// TIA Portal project "Trabajo_plantilla" (V14)
// Plantilla para la realización de la parte de programación de la asignatura de Automatización

(* hardware
DEVICE "S71500/ET200MP station_1"  S7-1500 station
   slot 0: "Perfil soporte_0"  Rack  6ES7 590-1***0-0AA0
   slot 1: "FINAL"  CPU 1516F-3 PN/DP  6ES7 516-3FN00-0AB0  V1.8
      slot 3: "Display de la CPU_1"  6ES7591-1BA00-0AA0
   slot 2: "DI 32x24VDC HF_1"  DI 32x24VDC HF  6ES7 521-1BL00-0AB0  V2.1
   slot 3: "DQ 16x24VDC/0.5A HF_1"  DQ 16x24VDC/0.5A HF  6ES7 522-1BH01-0AB0  V1.0
   slot 4: "AI 8xU/I/RTD/TC ST_1"  AI 8xU/I/RTD/TC ST  6ES7 531-7KF00-0AB0  V2.1
   slot 5: "AQ 4xU/I ST_1"  AQ 4xU/I ST  6ES7 532-5HD00-0AB0  V2.1
   slot 6: "DI 32x24VDC HF_2"  DI 32x24VDC HF  6ES7 521-1BL00-0AB0  V2.1
*)

// ===== PLC "FINAL"  CPU 1516F-3 PN/DP =====

VAR_GLOBAL   // PLC tag table "Variables maq_tem_HORNO"
   "Rearme_HORNO" AT %E2.1 : Bool;
   "Emer_HORNO" AT %E2.2 : Bool;
   "T_Cinta_Horno" AT %T8 : Timer;
   "Temperatura_REAL_HORNO" AT %MD11 : Real;
   "Temperatura_SENSOR_HORNO" AT %EW10 : Int;
   "Aviso_Foco_OK_HORNO" AT %M2.2 : Bool;
   "Aviso_error_sincrono_EXT_HORNO" AT %M2.4 : Bool;
   "Aviso_error_sensor_EXT_HORNO" AT %M2.5 : Bool;
   "S_piezas_cargadas_HORNO" AT %E2.3 : Bool;
   "S_piezas_descargadas_HORNO" AT %E2.4 : Bool;
   "MOV_CINTA_HORNO" AT %A0.0 : Bool;
   "FOCO_HORNO" AT %A2.2 : Bool;
   "MODO_FOCO" AT %E2.5 : Bool;
   "Aviso_Standby_HORNO" AT %M2.6 : Bool;
   "START_HORNO" AT %E2.0 : Bool;
END_VAR

VAR_GLOBAL   // PLC tag table "Variables CONFORMADORA"
   "Emer_CONFOR" AT %E1.2 : Bool;
   "Rearme_CONFOR" AT %E1.1 : Bool;
   "S_final_CONFOR" AT %E1.3 : Bool;
   "T_compresion_CONFOR" AT %T1 : Timer;
   "T_descompresion_CONFOR" AT %T2 : Timer;
   "Fuerza_SENSOR_CONFOR" AT %EW12 : Int;
   "Aviso_Pieza_Cargada_CONFOR" AT %E1.4 : Bool;
   "Aviso_Pieza_Desargada_CONFOR" AT %E1.5 : Bool;
   "Aviso_Standby_CONFOR" AT %M1.0 : Bool;
   "Aviso_error_sincrono_EXT_CONFOR" AT %M1.1 : Bool;
   "Aviso_error_sensor_EXT_CONFOR" AT %M1.2 : Bool;
   "Fuerza_REAL_CONFOR" AT %MD7 : Real;
   "COMPRIMIR_CONFOR" AT %A1.0 : Bool;
   "DESCOMPRIMIR_CONFOR" AT %A1.1 : Bool;
   "START_CONFOR" AT %E1.0 : Bool;
END_VAR

VAR_GLOBAL   // PLC tag table "Variables ROBOT"
   "START_ROBOT" AT %E5.0 : Bool;
   "EMER_ROBOT" AT %E5.1 : Bool;
   "Rearme_ROBOT" AT %E5.3 : Bool;
   "Tlimite_ROBOT" AT %T11 : Timer;
   "T_espera_ROBOT" AT %T12 : Timer;
   "MODO_M1_Descarga_ROBOT" AT %M5.0 : Bool;
   "MODO_M2_Carga_ROBOT" AT %M5.1 : Bool;
   "Zona_descarga_libre" AT %M5.2 : Bool;
   "Aviso_error_sincrono_ROBOT" AT %M5.3 : Bool;
   "Aviso_error_asincrono_ROBOT" AT %M5.4 : Bool;
   "Aviso_emergencia_ROBOT" AT %M5.5 : Bool;
   "Aviso_de_standby_ROBOT" AT %M5.6 : Bool;
   "SB_pieza_esperando" AT %E5.4 : Bool;   // Variables brazo robot
   "SB_pinza_llena_brazo" AT %E5.5 : Bool;
   "SB_llegada_Carga" AT %E5.6 : Bool;
   "SB_llegada_Descarga" AT %E5.7 : Bool;
   "SB_llegada_a_reposo" AT %E5.2 : Bool;
   "Mov1" AT %A5.0 : Bool;
   "Mov2" AT %A5.1 : Bool;
   "Mov3" AT %A5.2 : Bool;
   "Act1" AT %A5.3 : Bool;
   "Act2" AT %A5.4 : Bool;
   "X_Espera_maquina_libre" AT %M5.7 : Bool;
   "Aviso_STDBY_ROBOT" AT %M6.0 : Bool;
   "Aviso_maquina_libre" AT %M6.1 : Bool;
END_VAR

VAR_GLOBAL   // PLC tag table "Variables maq_tem_TUNEL"
   "Rearme_TUNEL" AT %E3.1 : Bool;
   "Emer_TUNEL" AT %E3.2 : Bool;
   "T_Cinta_Tunel" AT %T9 : Timer;
   "Temperatura_REAL_TUNEL" AT %MD15 : Real;
   "Temperatura_SENSOR_TUNEL" AT %EW8 : Int;
   "Aviso_Foco_OK_TUNEL" AT %M3.1 : Bool;
   "Aviso_error_sincrono_EXT_TUNEL" AT %M3.3 : Bool;
   "Aviso_error_sensor_EXT_TUNEL" AT %M3.4 : Bool;
   "S_piezas_descargadas_TUNEL" AT %E3.4 : Bool;
   "MOV_CINTA_TUNEL" AT %A3.0 : Bool;
   "FOCO_TUNEL" AT %A3.1 : Bool;
   "MODO_FOCO_TUNEL" AT %E3.5 : Bool;
   "Aviso_Standby_TUNEL" AT %M3.5 : Bool;
   "START_TUNEL" AT %E3.0 : Bool;
   "S_piezas_cargadas_TUNEL" AT %E3.3 : Bool;
END_VAR

VAR_GLOBAL   // PLC tag table "Variables PULIDORA"
   "Spieza_PULI" AT %E6.0 : Bool;
   "S_F_Mov_Cab" AT %E6.1 : Bool;
   "S_F_Mov_Cab2" AT %E6.2 : Bool;
   "S_F_Acercar" AT %E6.3 : Bool;
   "S_F_Pulido1" AT %E6.4 : Bool;
   "S_F_Pulido2" AT %E6.5 : Bool;
   "S_F_Cambio" AT %E6.6 : Bool;
   "S_F_Alejar" AT %E6.7 : Bool;
   "S_F_Giro" AT %E7.0 : Bool;
   "S_F_Giro2" AT %E7.1 : Bool;
   "T_Mov_Cab" AT %T13 : Timer;
   "T_Mov_Cab2" AT %T14 : Timer;
   "T_Acercar" AT %T15 : Timer;
   "T_Pulido1" AT %T16 : Timer;
   "T_Pulido2" AT %T17 : Timer;
   "T_Cambio" AT %T18 : Timer;
   "T_Alejar" AT %T19 : Timer;
   "T_Giro" AT %T20 : Timer;
   "T_Giro2" AT %T21 : Timer;
   "Bdf_Mov_Cab" AT %M9.6 : Bool;
   "Bdf_Mov_Cab2" AT %M9.7 : Bool;
   "Bdf_Acercar" AT %M14.0 : Bool;
   "Bdf_Alejar" AT %M14.1 : Bool;
   "Bdf_Giro1" AT %M14.2 : Bool;
   "Bdf_Giro2" AT %M14.3 : Bool;
   "Bdf_Pulido1" AT %M14.4 : Bool;
   "Bdf_Pulido2" AT %M14.5 : Bool;
   "Bdf_Cambio" AT %M14.6 : Bool;
   "Error_MovCab_T" AT %M14.7 : Bool;
   "Error_MovCab2_T" AT %M15.0 : Bool;
   "Error_Acercar_T" AT %M15.1 : Bool;
   "Error_Pulido_T1" AT %M15.2 : Bool;
   "Error_Pulido2_T" AT %M15.3 : Bool;
   "Error_Cambio_T" AT %M15.4 : Bool;
   "Error_Alejar_T" AT %M15.5 : Bool;
   "Error_Giro_T" AT %M15.6 : Bool;
   "Error_Giro2_T" AT %M15.7 : Bool;
   "Mover_Cabezal1" AT %A7.0 : Bool;
   "Mover_Cabezal2" AT %A7.1 : Bool;
   "Acercar" AT %A7.2 : Bool;
   "Pulido1" AT %A7.3 : Bool;
   "Pulido2" AT %A7.4 : Bool;
   "Cambio" AT %A7.5 : Bool;
   "Alejar" AT %A7.6 : Bool;
   "Giro_Soporte1" AT %A7.7 : Bool;
   "Giro_Soporte2" AT %A8.0 : Bool;
   "Aviso_Error_Asinc_PULI" AT %M4.0 : Bool;
   "Aviso_Error_Sinc_PULI" AT %M4.1 : Bool;
   "EMER_PULI" AT %E7.3 : Bool;
   "REARME_PULI" AT %E7.4 : Bool;
   "Aviso_StdBy_PULI" AT %M4.2 : Bool;
   "START_PULI" AT %E7.2 : Bool;
END_VAR

VAR_GLOBAL   // PLC tag table "Variables_GENERAL"
   "ON" AT %E0.0 : Bool;
   "EMER" AT %E0.1 : Bool;
   "Rearme" AT %E0.2 : Bool;
   "MA" AT %E0.3 : Bool;
   "MB" AT %E0.4 : Bool;
   "X0" AT %M0.0 : Bool;
   "X1" AT %M0.1 : Bool;
   "X2" AT %M0.2 : Bool;
   "X3" AT %M0.3 : Bool;
   "X4" AT %M0.4 : Bool;
   "X5" AT %M0.5 : Bool;
   "X_CONFORMADO" AT %M6.2 : Bool;
   "X_HORNO" AT %M6.3 : Bool;
   "X_TUNEL" AT %M6.4 : Bool;
   "X_PULIDORA" AT %M6.5 : Bool;
   "X_ROBOT" AT %M6.6 : Bool;
   "X20_Marcha" AT %M20.0 : Bool;
   "X21_EMER" AT %M20.1 : Bool;
   "X10_GMM" AT %M20.2 : Bool;
   "X11_MMA" AT %M20.3 : Bool;
   "X12_MMB" AT %M20.4 : Bool;
   "mfON" AT %E0.5 : Bool;
END_VAR

DATA_BLOCK "DATOS_PRODUCCION"   // DB1
TITLE = parametros de produccion (TODOS)
{ S7_Optimized_Access := 'TRUE' }
VERSION : 0.1
// Incluye cualquier  constante numérica necesaria para el control. Este bloque se podría descomponer en varios bloques de datos temáticos si fuera necesario.
   VAR
      HI_LIM : Real := 1000.0;
      LOW_LIM : Real := 0.0;
      Fuerza_necesaria_CONFOR : Real;
      Tiempo_lim_CONFOR : S5Time := S5T#30s;   // T. max de maniobra para la prensa
      Tiempo_lim_Cinta_Horno : S5Time := S5T#30s;   // Tiempo limite de maniobra para el sistema de carga interno del torno
      Tiempo_lim_Cinta_Tunel : S5Time := S5T#30s;   // T. lim. de la maniobra abrir o cerrar compuerta para el torno
      Temperatura_OK_HORNO : Real;
      Temperatura_OK_TUNEL : Real;
      Temperatura_lim_HORNO : Real := 800.0;   // Fuerza que se debe realizar la prensa (kN)
      Temperatura_lim_TUNEL : Real := 5.0;   // Fuerza que se debe realizar la prensa (kN)
      T_PULI_Giro : S5Time := S5T#20s;
      T_PULI_Mov_Puli : S5Time := S5T#20s;
      T_PULI_Pulido : S5Time;
      T_PULI_Cambio : S5Time := S5T#20s;
      Tiempo_lim_brazo : S5Time := S5T#5m;
   END_VAR
BEGIN
END_DATA_BLOCK

DATA_BLOCK "DATOS_PRODUCCION_MODO_B"   // DB3
TITLE = parametros de producción MODO_A
{ S7_Optimized_Access := 'TRUE' }
VERSION : 0.1
// subconjunto de parámetros de DATOS_PRODUCCION (DB1)
   VAR
      Fuerza_necesaria_CONFOR : Real := 900.0;   // Fuerza a realizar por la prensa (kN)
      Temperatura_necesaria_HORNO : Real := 700.0;
      Temperatura_necesaria_TUNEL : Real := 10.0;
      Tiempo_lim_PULIDO : S5Time := S5T#90s;
   END_VAR
BEGIN
END_DATA_BLOCK

DATA_BLOCK "DATOS_PRODUCCION_MODO_A"   // DB4
TITLE = parametros de producción MODO_A
{ S7_Optimized_Access := 'TRUE' }
VERSION : 0.1
// subconjunto de parámetros de DATOS_PRODUCCION (DB1)
   VAR
      Fuerza_necesaria_CONFOR : Real := 700.0;   // Fuerza a realizar por la prensa (kN)
      Temperatura_necesaria_HORNO : Real := 600.0;
      Temperatura_necesaria_TUNEL : Real := 15.0;
      Tiempo_lim_PULIDO : S5Time := S5T#30s;
   END_VAR
BEGIN
END_DATA_BLOCK

// folder: maquinas

DATA_BLOCK "CONFORMADORA_DB"   // DB7
{ S7_Optimized_Access := 'TRUE' }
VERSION : 0.1
// stored: InstanceOfName CONFORMADORA
"CONFORMADORA"
BEGIN
END_DATA_BLOCK

DATA_BLOCK "maq_temp_DB_TUNEL"   // DB9
{ S7_Optimized_Access := 'TRUE' }
VERSION : 0.1
// stored: InstanceOfName maq_temp
"maq_temp"
BEGIN
END_DATA_BLOCK

DATA_BLOCK "ROBOT_DB"   // DB11
{ S7_Optimized_Access := 'TRUE' }
VERSION : 0.1
// stored: InstanceOfName ROBOT
"ROBOT"
BEGIN
END_DATA_BLOCK

DATA_BLOCK "maq_temp_DB_HORNO"   // DB13
{ S7_Optimized_Access := 'TRUE' }
VERSION : 0.1
// stored: InstanceOfName maq_temp
"maq_temp"
BEGIN
END_DATA_BLOCK

DATA_BLOCK "PULIDORA_DB"   // DB15
{ S7_Optimized_Access := 'TRUE' }
VERSION : 0.1
// stored: InstanceOfName PULIDORA
"PULIDORA"
BEGIN
END_DATA_BLOCK

// folder: (top level)

ORGANIZATION_BLOCK "Main"   // OB1, LAD, ProgramCycle
TITLE = "Main Program Sweep (Cycle)"
{ S7_Optimized_Access := 'TRUE' }
VERSION : 0.1
// Contenido del  Programa Principal:
// A)  Segmentos con llamadas incondicionales a otros bloques por orden de prioridad (GEMER, MODOS DE MARCHA, FLANCOS y CONECTORES, ANALOGICA ,  bloques TIPO MÁQUINA) .
// 
// B) Resto de segmentos
   VAR_INPUT
      Initial_Call : Bool;   // Initial call of this OB
      Remanence : Bool;   // =True, if remanent data are available
   END_VAR
BEGIN

REGION Network 1 (STL): Llamada a tests unitarios
   //    CALL  "test_trat_sensor_temperatura"
   //    CALL  "test_COMFORMADORA"
   //    CALL  "test_maq_temp"
   //    CALL  "test_PULIDORA"
   //    CALL  "test_ROBOT"
END_REGION

REGION Network 2 (STL): Llamadas incondicionales a bloques
         CALL  "grafcet_modos_de_marcha";
         CALL  "grafcet_seguridad";
END_REGION

REGION Network 3 (STL): Activación de la producción en la celda
         A     "X0";

         A(;
         A     "ON";
         FP    "mfON";
         );

         A(;
         O     "X11_MMA";
         O     "X12_MMB";
         );

         R     "X0";
         S     "X1";
         S     "X2";
         S     "X3";
         S     "X4";
         S     "X5";
END_REGION

REGION Network 4 (STL): paso de etapas de espera a unidades productivas
   // Encendido de las unidades productivas
         A     "X1";
         A     "START_CONFOR";
         S     "X_CONFORMADO";
         R     "X1";

         A     "X2";
         A     "START_HORNO";
         S     "X_HORNO";
         R     "X2";


         A     "X3";
         A     "START_TUNEL";
         S     "X_TUNEL";
         R     "X3";

         A     "X4";
         A     "START_PULI";
         S     "X_PULIDORA";
         R     "X4";

         A     "X5";
         A     "START_ROBOT";
         A(;
         O     "MODO_M1_Descarga_ROBOT";
         O     "MODO_M2_Carga_ROBOT";
         );
         S     "X_ROBOT";
         R     "X5";
END_REGION

REGION Network 5 (STL): Tratamiento de estación CONFORMADORA
         A     "X_CONFORMADO";
         JCN   _LLAMADA_COMFORMADORA;

         CALL  "CONFORMADORA", "CONFORMADORA_DB"
         ( START                    := "START_CONFOR",
           REARME                   := "Rearme_CONFOR",
           EMER                     := "Emer_CONFOR",
           S_fin                    := "S_final_CONFOR",
           Tiempo_MAX_maniobra      := "DATOS_PRODUCCION".Tiempo_lim_CONFOR,
           Temp_Ciclo_compre        := "T_compresion_CONFOR",
           Temp_Ciclo_descompre     := "T_descompresion_CONFOR",
           Fuerza_SENSOR            := "Fuerza_SENSOR_CONFOR",
           HI_LIM                   := "DATOS_PRODUCCION".HI_LIM,
           LO_LIM                   := "DATOS_PRODUCCION".LOW_LIM,
           Aviso_Pieza_Cargada      := "Aviso_Pieza_Cargada_CONFOR",
           Aviso_Pieza_Descargada   := "Aviso_Pieza_Desargada_CONFOR",
           FUERZA_NECESARIA         := "DATOS_PRODUCCION".Fuerza_necesaria_CONFOR,
           COMPRIMIR                := "COMPRIMIR_CONFOR",
           DESCOMPRIR               := "DESCOMPRIMIR_CONFOR",
           Aviso_Standby            := "Aviso_Standby_CONFOR",
           Aviso_error_sincrono_EXT := "Aviso_error_sincrono_EXT_CONFOR",
           Aviso_error_sensor_EXT   := "Aviso_error_sensor_EXT_CONFOR",
           FUERZA_REAL              := "Fuerza_REAL_CONFOR"
         );

   _LLAMADA_COMFORMADORA:NOP   0;

         A     "X_CONFORMADO";
         AN    "START_CONFOR";
         R     "X_CONFORMADO";
         S     "X1";
END_REGION

REGION Network 6 (STL): Tratamiento de estación HORNO
         A     "X_HORNO";
         JCN   _LLAMADA_HORNO;

         CALL  "maq_temp", "maq_temp_DB_HORNO"
         ( START                    := "START_HORNO",
           REARME                   := "Rearme_HORNO",
           EMER                     := "Emer_HORNO",
           Tiempo_MAX_maniobra      := "DATOS_PRODUCCION".Tiempo_lim_Cinta_Horno,
           Tempo_maniobra           := "T_Cinta_Horno",
           Temperatura_SENSOR       := "Temperatura_SENSOR_HORNO",
           HI_LIM                   := "DATOS_PRODUCCION".HI_LIM,
           LO_LIM                   := "DATOS_PRODUCCION".LOW_LIM,
           Modo_Foco                := TRUE,
           Aviso_Piezas_Cargadas    := "S_piezas_cargadas_HORNO",
           Aviso_Piezas_Descargadas := "S_piezas_descargadas_HORNO",
           Temperatura_limite       := "DATOS_PRODUCCION".Temperatura_lim_HORNO,
           Temperatura_OK           := "DATOS_PRODUCCION".Temperatura_OK_HORNO,
           FOCO                     := "FOCO_HORNO",
           MOV                      := "MOV_CINTA_HORNO",
           Aviso_OK                 := "Aviso_Foco_OK_HORNO",
           Aviso_Standby            := "Aviso_Standby_HORNO",
           Aviso_error_sincrono_EXT := "Aviso_error_sincrono_EXT_HORNO",
           Aviso_error_sensor_EXT   := "Aviso_error_sensor_EXT_HORNO",
           Temperatura_REAL         := "Temperatura_REAL_HORNO"
         );

   _LLAMADA_HORNO:NOP   0;

         A     "X_HORNO";
         AN    "START_HORNO";
         R     "X_HORNO";
         S     "X2";
END_REGION

REGION Network 7 (STL): Tratamiento de estación TUNEL
         A     "X_TUNEL";
         JCN   _LLAMADA_TUNEL;


         CALL  "maq_temp","maq_temp_DB_TUNEL"
         ( START                    := "START_TUNEL",
           REARME                   := "Rearme_TUNEL",
           EMER                     := "Emer_TUNEL",
           Tiempo_MAX_maniobra      := "DATOS_PRODUCCION".Tiempo_lim_Cinta_Tunel,
           Tempo_maniobra           := "T_Cinta_Tunel",
           Temperatura_SENSOR       := "Temperatura_SENSOR_TUNEL",
           HI_LIM                   := "DATOS_PRODUCCION".HI_LIM,
           LO_LIM                   := "DATOS_PRODUCCION".LOW_LIM,
           Modo_Foco                := FALSE,
           Aviso_Piezas_Cargadas    := "S_piezas_cargadas_TUNEL",
           Aviso_Piezas_Descargadas := "S_piezas_descargadas_TUNEL",
           Temperatura_limite       := "DATOS_PRODUCCION".Temperatura_lim_TUNEL,
           Temperatura_OK           := "DATOS_PRODUCCION".Temperatura_OK_TUNEL,
           FOCO                     := "FOCO_TUNEL",
           MOV                      := "MOV_CINTA_TUNEL",
           Aviso_OK                 := "Aviso_Foco_OK_TUNEL",
           Aviso_Standby            := "Aviso_Standby_TUNEL",
           Aviso_error_sincrono_EXT := "Aviso_error_sincrono_EXT_TUNEL",
           Aviso_error_sensor_EXT   := "Aviso_error_sensor_EXT_TUNEL",
           Temperatura_REAL         := "Temperatura_REAL_TUNEL"
         );

   _LLAMADA_TUNEL:NOP   0;

         A     "X_TUNEL";
         AN    "START_TUNEL";
         R     "X_TUNEL";
         S     "X3";
END_REGION

REGION Network 8 (STL): Tratamiento de estación PULIDORA
         A     "X_PULIDORA";
         JCN   _LLAMADA_PULIDORA;

         CALL  "PULIDORA", "PULIDORA_DB"
         ( Spieza                := "Spieza_PULI",
           SFMovCab              := "S_F_Mov_Cab",
           SFMovCab2             := "S_F_Mov_Cab2",
           SF_Acercar            := "S_F_Acercar",
           SFPulido1             := "S_F_Pulido1",
           SFPulido2             := "S_F_Pulido2",
           SFCambio              := "S_F_Cambio",
           SFAlejar              := "S_F_Alejar",
           SFGiro                := "S_F_Giro",
           SFGiro2               := "S_F_Giro2",
           T_Max_MovCab          := "DATOS_PRODUCCION".T_PULI_Pulido,
           T_Max_Mov_Cab2        := "DATOS_PRODUCCION".T_PULI_Pulido,
           T_Max_Acercar         := "DATOS_PRODUCCION".T_PULI_Mov_Puli,
           T_Max_Pulido          := "DATOS_PRODUCCION".T_PULI_Pulido,
           T_Max_Pulido2         := "DATOS_PRODUCCION".T_PULI_Pulido,
           T_Max_Cambio          := "DATOS_PRODUCCION".T_PULI_Cambio,
           T_Max_Alejar          := "DATOS_PRODUCCION".T_PULI_Mov_Puli,
           T_Max_Giro            := "DATOS_PRODUCCION".T_PULI_Giro,
           T_Max_Giro2           := "DATOS_PRODUCCION".T_PULI_Giro,
           TMovCab               := "T_Mov_Cab",
           TMovCab2              := "T_Mov_Cab2",
           TAcercar              := "T_Acercar",
           TPulido1              := "T_Pulido1",
           TPulido2              := "T_Pulido2",
           TCambio               := "T_Cambio",
           TAlejar               := "T_Alejar",
           TGiro                 := "T_Giro",
           TGiro2                := "T_Giro2",
           START                 := "START_PULI",
           REARME                := "REARME_PULI",
           EMER                  := "EMER_PULI",
           Mover_Cabezal         := "Mover_Cabezal1",
           Mover_Cabezal2        := "Mover_Cabezal2",
           Acercar_              := "Acercar",
           Pulido_               := "Pulido1",
           Cambio_               := "Cambio",
           Pulido2_              := "Pulido2",
           Alejar_               := "Alejar",
           Giro_                 := "Giro_Soporte1",
           Giro2                 := "Giro_Soporte2",
           Aviso_StandBy         := "Aviso_StdBy_PULI",
           Aviso_Error_Asíncrono := "Aviso_Error_Asinc_PULI",
           Aviso_Error_Sincrono  := "Aviso_Error_Sinc_PULI"
         );

   _LLAMADA_PULIDORA:NOP   0;

         A     "X_PULIDORA";
         AN    "START_PULI";
         R     "X_PULIDORA";
         S     "X4";
END_REGION

REGION Network 9 (STL): Tratamiento de estación ROBOT
         A     "X_ROBOT";
         JCN   _LLAMADA_ROBOT;

         CALL  "ROBOT", "ROBOT_DB"
         ( Sensor_Pieza            := "SB_pieza_esperando",
           Sensor_Pinza_Llena      := "SB_pinza_llena_brazo",
           Sensor_Llegada_Carga    := "SB_llegada_Carga",
           Sensor_Llegada_Descarga := "SB_llegada_Descarga",
           Sensor_Llegada_a_Reposo := "SB_llegada_a_reposo",
           START                   := "START_ROBOT",
           EMER                    := "EMER_ROBOT",
           REARME                  := "Rearme_ROBOT",
           Tiempo_lim              := "DATOS_PRODUCCION".Tiempo_lim_brazo,
           Timer_LIM               := "Tlimite_ROBOT",
           X_Marcha_1              := "MODO_M1_Descarga_ROBOT",
           X_Marcha_2              := "MODO_M2_Carga_ROBOT",
           Mov1                    := "Mov1",
           Mov2                    := "Mov2",
           Mov3                    := "Mov3",
           Act1                    := "Act1",
           Act2                    := "Act2",
           Wait                    := "X_Espera_maquina_libre",
           Aviso_Emergencia        := "Aviso_emergencia_ROBOT",
           STDBY                   := "Aviso_STDBY_ROBOT",
           Aviso_Maquina_Libre     := "Aviso_maquina_libre",
           Aviso_Error_Sincrono    := "Aviso_error_sincrono_ROBOT",
           Aviso_Error_Asincrono   := "Aviso_error_asincrono_ROBOT"
         );

   _LLAMADA_ROBOT:NOP   0;

         A     "X_ROBOT";
         AN    "START_ROBOT";
         R     "X_ROBOT";
         S     "X5";
END_REGION
END_ORGANIZATION_BLOCK

ORGANIZATION_BLOCK "Startup"   // OB100, LAD, Startup
TITLE = "Complete Restart"
{ S7_Optimized_Access := 'TRUE' }
VERSION : 0.1
// Bloque de arranque: se ejecuta una única vez antes del bloque OB1
   VAR_INPUT
      LostRetentive : Bool;   // True if retentive data are lost
      LostRTC : Bool;   // True if date and time are lost
   END_VAR
BEGIN

REGION Network 1 (STL): ARRANQUE
         SET;
         S     "X0";
         S     "X20_Marcha";
         S     "X10_GMM";

         R     "X1";
         R     "X2";
         R     "X3";
         R     "X4";
         R     "X5";
         R     "X_CONFORMADO";
         R     "X_HORNO";
         R     "X_TUNEL";
         R     "X_PULIDORA";
         R     "X_ROBOT";

   //METACONTROL
         R     "X21_EMER";
         R     "X11_MMA";
         R     "X12_MMB";

   //L     DW#16#0
   //T     "Tag_1"              //MD10 marcas desde %M10.0 a %MD13.7

         R     "mfON";

   //R estados que no corresponden al reposo
   //S estados que corresponden al reposo
END_REGION
END_ORGANIZATION_BLOCK

// folder: analógico

FUNCTION "TRAT_SENSOR_TEMPERATURA" : Void   // FC2, LAD
{ S7_Optimized_Access := 'TRUE' }
VERSION : 0.1
   VAR_INPUT
      RAW : Int;   // Valor del transductor muestreado
      BIPOLAR : Bool;   // TRUE +- 27.648 valores, FALSE +27.648 valores
      HI_LIM : Real;
      LO_LIM : Real;
      Temperatura_limite : Real;
      Temperatura_OK : Real;
      Modo_FOCO : Bool;
      RESET : Bool;   // Salidas a nivel bajo. Salida de bloque
   END_VAR
   VAR_OUTPUT
      Aviso_Foco_encendido : Bool;
      Aviso_Foco_OK : Bool;
   END_VAR
   VAR_IN_OUT
      Error : Bool;   // Valor medido en máximos o mínimos del campo de trabajo
      Real_Val : Real;
   END_VAR
   VAR_TEMP
      retSCALE : Word;   // W#16#0000 si no hay fallos y W#16#0008 si los hay
      Aviso_tem_OK_Horno : Bool;
      Aviso_tem_OK_Tunel : Bool;
      Aviso_encendido_Horno : Bool;
      Aviso_encendido_Tunel : Bool;
   END_VAR
BEGIN

REGION Network 1 (STL): RESET
         A     #RESET;
         R     #Error;
         R     #Aviso_Foco_OK;

         JCN   _RES;
         L     0.0;
         T     #Real_Val;  //transfieres el valor 0.0 a la variable #REAL_VAL
   _RES: NOP   0;

   //Volver a cagar la señal de RESET, pues el RLO ha sido modificado a TRUE por el salto
         A     #RESET;
         BEC;
END_REGION

REGION Network 2: LLAMADA A SCALE
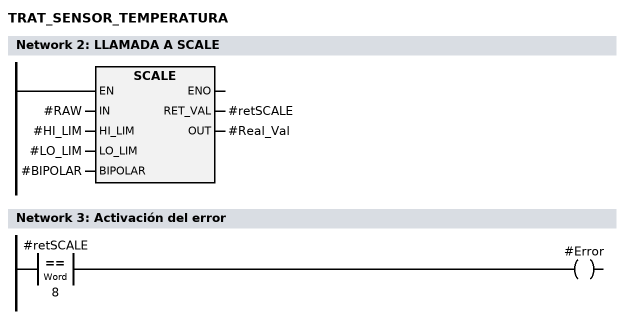
   #retSCALE := SCALE(IN := #RAW, HI_LIM := #HI_LIM, LO_LIM := #LO_LIM, BIPOLAR := #BIPOLAR, OUT => #Real_Val);
END_REGION

REGION Network 3: Activación del error
   RUNG wire#powerrail
      { S7_Templates := "SrcType := Word" } EQ_Contact(in1 := #retSCALE, in2 := 8)
      Coil( #Error )
   END_RUNG
   // the same network as SCL:
   #Error := #retSCALE = 8;
END_REGION

REGION Network 4 (STL): Tratamiento aviso de temperatura limite en Horno/Tunel
         L     #Real_Val;
         L     #Temperatura_limite;
         >R;
         R     #Aviso_encendido_Horno;
         S     #Aviso_encendido_Tunel;
END_REGION

REGION Network 5 (STL): "
         A     <=0;
         S     #Aviso_encendido_Horno;
         R     #Aviso_encendido_Tunel;
END_REGION

REGION Network 6 (STL): Tratamiento aviso de temperatura OK en Horno/Tunel
         L     #Real_Val;
         L     #Temperatura_OK;
         >R;
         S     #Aviso_tem_OK_Horno;
         R     #Aviso_tem_OK_Tunel;
END_REGION

REGION Network 7 (STL): "
         A     <=0;
         R     #Aviso_tem_OK_Horno;
         S     #Aviso_tem_OK_Tunel;
END_REGION

REGION Network 8 (STL)
         A     #Modo_FOCO;
         JCN   _FOCO;

         A     #Aviso_encendido_Horno;
         =     #Aviso_Foco_encendido;

         A     #Aviso_tem_OK_Horno;
         =     #Aviso_Foco_OK;

   _FOCO:NOP   0;
END_REGION

REGION Network 9 (STL)
         AN    #Modo_FOCO;
         JCN   _TUNEL;

         A     #Aviso_encendido_Tunel;
         =     #Aviso_Foco_encendido;


         A     #Aviso_tem_OK_Tunel;
         =     #Aviso_Foco_OK;

   _TUNEL:NOP   0;
END_REGION

REGION Network 10 (STL): EN-ENO compliant
   // Pone el biestale RB a FALSE si hay un ERROR síncrono. En este caso esto implica que hay un error en la medida
         AN    #Error;
         SAVE;  // RB := RLO
END_REGION
END_FUNCTION

FUNCTION "TRAT_SENSOR_FUERZA" : Void   // FC8, LAD
{ S7_Optimized_Access := 'TRUE' }
VERSION : 0.1
   VAR_INPUT
      RAW : Int;   // Valor del transductor muestreado
      BIPOLAR : Bool;   // TRUE +- 27.648 valores, FALSE +27.648 valores
      HI_LIM : Real;
      LO_LIM : Real;
      FUERZA_NECESARIA : Real;   // Fuerza a realizar
      RESET : Bool;   // Salidas a nivel bajo. Salida de bloque
   END_VAR
   VAR_OUTPUT
      Aviso_Fuerza_Necesaria : Bool;   // True si fuerza >=FUERZA_NECESARIA
   END_VAR
   VAR_IN_OUT
      Error : Bool;   // Valor medido en máximos o mínimos del campo de trabajo
      Real_Val : Real;
   END_VAR
   VAR_TEMP
      retSCALE : Word;   // W#16#0000 si no hay fallos y W#16#0008 si los hay
   END_VAR
BEGIN

REGION Network 1 (STL): RESET
         A     #RESET;
         R     #Error;
         R     #Aviso_Fuerza_Necesaria;

         JCN   _RES;
         L     0.0;
         T     #Real_Val;  //transfieres el valor 0.0 a la variable #REAL_VAL
   _RES: NOP   0;

   //Volver a cagar la señal de RESET, pues el RLO ha sido modificado a TRUE por el salto
         A     #RESET;
         BEC;
END_REGION

REGION Network 2: LLAMADA A SCALE
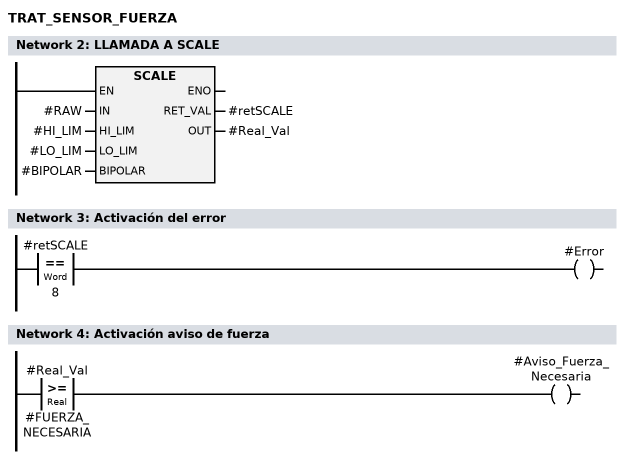
   #retSCALE := SCALE(IN := #RAW, HI_LIM := #HI_LIM, LO_LIM := #LO_LIM, BIPOLAR := #BIPOLAR, OUT => #Real_Val);
END_REGION

REGION Network 3: Activación del error
   RUNG wire#powerrail
      { S7_Templates := "SrcType := Word" } EQ_Contact(in1 := #retSCALE, in2 := 8)
      Coil( #Error )
   END_RUNG
   // the same network as SCL:
   #Error := #retSCALE = 8;
END_REGION

REGION Network 4: Activación aviso de fuerza
   RUNG wire#powerrail
      { S7_Templates := "SrcType := Real" } GE_Contact(in1 := #Real_Val, in2 := #FUERZA_NECESARIA)
      Coil( #Aviso_Fuerza_Necesaria )
   END_RUNG
   // the same network as SCL:
   #Aviso_Fuerza_Necesaria := #Real_Val >= #FUERZA_NECESARIA;
END_REGION

REGION Network 5 (STL): EN-ENO compliant
   // Pone el biestale RB a FALSE si hay un ERROR síncrono. En este caso esto implica que hay un error en la medida
         AN    #Error;
         SAVE;  // RB := RLO
END_REGION
END_FUNCTION

// folder: maniobras

FUNCTION_BLOCK "MOV_BRAZO_1"   // FB1, STL
{ S7_Optimized_Access := 'TRUE' }
VERSION : 0.1
// Maniobra para cuando el robot tiene que realizar una carga o un descarga en una maquina. Incluye  la carga y descarga de la pieza y la espera hasta que la máquina este descargada para poder introducir la pieza
   VAR_INPUT
      Sensor_Pieza : Bool;   // Sensor que detecta si hay una pieza que el robot tiene que coger
      Sensor_Pinza_Llena : Bool;   // Sensor que detecta si la pinza tiene una pieza o no
      Sensor_Llegada_a_Buffer : Bool;   // Sensor que detecta que el robot ha llegado al buffer
      Sensor_Llegada_a_Maquina : Bool;   // Sensor que detecta la llegada del robot a la máquina
      "Sensor_Llegada_a _Reposo" : Bool;   // Sensor que detecta la llegada del robot a la posición de reposo
      EMER : Bool;   // Entrada que indica la entrada del sistema en emergencia
      Tiempo_lim : S5Time;   // Tiempo limite de maniobra
      Timer_LIM : Timer;   // Temporizador para el tiempo limite de maniobra
   END_VAR
   VAR_OUTPUT
      MOV1 : Bool;   // Brazo se mueve a buffer
      MOV2 : Bool;   // Brazo se mueve a maquina
      MOV3 : Bool;   // Brazo se mueve a reposo
      ACT1 : Bool;   // Brazo coje pieza
      ACT2 : Bool;   // Brazo descarga pieza
      WAIT1 : Bool;   // Brazo espera a que la maquina este libre
   END_VAR
   VAR_IN_OUT
      Aviso_Error_Tiempo_Limite : Bool;   // Si se sobrepasa el tiempo se activa este aviso
      Aviso_Fin_Maniobra : Bool;   // Si la maniobra termina se activa este aviso para indicar que el brazo esta libre
      Aviso_Error_No_Pieza : Bool;   // Si no detecta una pieza cuando le han mandado a por una pieza el robot activa este error
      Aviso_Error_Pinza_Abierta : Bool;   // Si la pinza se abre en un momento que no deberia (MOV2 y WAIT1) se activa
      Aviso_Maquina_Libre : Bool;   // Aviso para indicar al robot que puede descargar en la maquina
   END_VAR
   VAR
      BDT : Bool;   // Bit de trabajo
      X1 : Bool;   // Etapa de MOV 1
      X2 : Bool;   // Etapa de ACT 1
      X3 : Bool;   // Etapa de MOV 2
      X4 : Bool;   // Etapa de WAIT
      X5 : Bool;   // Etapa de ACT2
      X6 : Bool;   // Etapa de MOV 3
      Aviso_Interno_Tiempo : Bool;   // Aviso interno de que ha psado el tiempo limite
      Aviso_Interno_FIN : Bool;   // Aviso intetno de fon de maniobra
      Aviso_Interno_Pinza_Abierta : Bool;   // Aviso interno de que la pinza esta abierta
      Aviso_Interno_NO_Pieza : Bool;   // Aviso interno de que no hay pieza
   END_VAR
BEGIN

REGION Network 1: DESCONEXIÓN RESET
   // MAX PRIORITY
         A     #EMER;
         R     #BDT;
         R     #Aviso_Error_No_Pieza;
         R     #Aviso_Error_Pinza_Abierta;
         R     #Aviso_Error_Tiempo_Limite;
         R     #Aviso_Fin_Maniobra;
         R     #MOV1;
         R     #MOV2;
         R     #MOV3;
         R     #ACT1;
         R     #ACT2;
         R     #WAIT1;

         R     #Timer_LIM;
         FR    #Timer_LIM;

         BEC;
END_REGION

REGION Network 2: DESCONEXION ERROR TIEMPO LIMITE
         A     #Aviso_Interno_Tiempo;
         R     #BDT;
         S     #Aviso_Error_Tiempo_Limite;
         R     #Aviso_Interno_Tiempo;
         R     #Timer_LIM;
         FR    #Timer_LIM;
         R     #MOV1;
         R     #MOV2;
         R     #MOV3;
         R     #ACT1;
         R     #ACT2;
         R     #WAIT1;

         BEC;
END_REGION

REGION Network 3: DESCONEXION ERROR NO PIEZA
         A     #Aviso_Interno_NO_Pieza;
         R     #BDT;
         S     #Aviso_Error_No_Pieza;
         R     #Aviso_Interno_NO_Pieza;
         R     #Timer_LIM;
         FR    #Timer_LIM;
         R     #MOV1;
         R     #MOV2;
         R     #MOV3;
         R     #ACT1;
         R     #ACT2;
         R     #WAIT1;



         BEC;
END_REGION

REGION Network 4: DESCONEXION ERROR PINZA ABIERTA
         A     #Aviso_Interno_Pinza_Abierta;
         R     #BDT;
         S     #Aviso_Error_Pinza_Abierta;
         R     #Aviso_Interno_Pinza_Abierta;
         R     #Timer_LIM;
         FR    #Timer_LIM;
         R     #MOV1;
         R     #MOV2;
         R     #MOV3;
         R     #ACT1;
         R     #ACT2;
         R     #WAIT1;



         BEC;
END_REGION

REGION Network 5: DESCONEXION FIN MANIOBRA
         A     #Aviso_Interno_FIN;
         R     #BDT;
         S     #Aviso_Fin_Maniobra;
         R     #Aviso_Interno_FIN;
         R     #Timer_LIM;
         FR    #Timer_LIM;
         R     #MOV1;
         R     #MOV2;
         R     #MOV3;
         R     #ACT1;
         R     #ACT2;
         R     #WAIT1;


         BEC;
END_REGION

REGION Network 6: CONEXION XMARCHA
         SET;
         L     #Tiempo_lim;
         SS    #Timer_LIM;
         FP    #BDT;

         S     #X1;
         R     #X2;
         R     #X3;
         R     #X4;
         R     #X5;
         R     #X6;
END_REGION

REGION Network 7: X1(Mov a BUFFER)->X2(captura de la pieza)
         A     #X1;
         A     #Sensor_Llegada_a_Buffer;  //sensor que indica he llegado al buffer
         S     #X2;  //Estado que simboliza carga de la pieza
         R     #X1;
END_REGION

REGION Network 8: X2(captura de la pieza)->X3 (Mov a maquina con pieza)
         A     #X2;
         A     #Sensor_Pinza_Llena;  //tengo objeto
         S     #X3;
         R     #X2;
END_REGION

REGION Network 9: X3(Mov a maquina con pieza)->X4(espera a maquina)
         A     #X3;
         A     #Sensor_Llegada_a_Maquina;  //llega a la maquina
         S     #X4;
         R     #X3;
END_REGION

REGION Network 10: X4 (espera a maquina ) -> X5(coloca pieza en maquina)
         A     #X4;
         A     #Aviso_Maquina_Libre;
         S     #X5;
         R     #X4;
END_REGION

REGION Network 11: X5(coloca pieza en máquina)->X6(Mov a reposo)
         A     #X5;
         AN    #Sensor_Pinza_Llena;
         S     #X6;
         R     #X5;
END_REGION

REGION Network 12: X6(Mov a reposo)->FIN
         A     #X6;
         A     #"Sensor_Llegada_a _Reposo";
         S     #Aviso_Interno_FIN;
         R     #X6;
         R     #Timer_LIM;
         FR    #Timer_LIM;
END_REGION

REGION Network 13: TRAT X1
         A     #X1;
         AN    #Sensor_Pieza;
         S     #Aviso_Interno_NO_Pieza;  //Significa que va a por una pieza y derrepente la pieza deja de estar.
   //Posible fallo de que el sensor no funcione o bien de pieza mal colocada, Requiere operario

         A     #X1;
         O;
         =     #MOV1;  //Indica que la máquina se mueve
END_REGION

REGION Network 14: TRAT X2
         A     #X2;
         =     #ACT1;
END_REGION

REGION Network 15: TRAT X3
         A     #X3;
         AN    #Sensor_Pinza_Llena;
         S     #Aviso_Interno_Pinza_Abierta;  //En el transporte la pinza de abre, la pieza se cae. ERROR GRAVE

         A     #X3;
         =     #MOV2;  //Indica que la máquina realiza el segundo movimiento
END_REGION

REGION Network 16: TRAT X4
         A     #X4;
         AN    #Sensor_Pinza_Llena;
         S     #Aviso_Interno_Pinza_Abierta;

         A     #X4;
         =     #WAIT1;

         A     #X4;
         R     #Timer_LIM;  //Se desactiva Timer ya que este estado depende del estado de la maquina
         FR    #Timer_LIM;
END_REGION

REGION Network 17: TRAT X5
         A     #X5;
         =     #ACT2;
END_REGION

REGION Network 18: TRAT X6
         A     #X6;
         =     #MOV3;
END_REGION

REGION Network 19: TRAT ERROR TIEMPO LIMITE
         A     #Timer_LIM;
         S     #Aviso_Error_Tiempo_Limite;
         R     #Timer_LIM;
         FR    #Timer_LIM;
END_REGION
END_FUNCTION_BLOCK

FUNCTION_BLOCK "MOV_CONFOR_FUERZA"   // FB4, STL
{ S7_Optimized_Access := 'TRUE' }
VERSION : 0.1
// Maniobra que permite tener un control de la fuerza del sensor y administra la salida
   VAR_INPUT
      Tiempo_Max_Ciclo : S5Time;   // tiempo maxino para que se reliace el ciclo
      Temp_Ciclo : Timer;   // Timer necesario para que se reliace el ciclo
      Fuerza_Bruta : Int;   // Señal analógica
      HI_LIM : Real;
      LO_LIM : Real;
      FUERZA_NECESARIA : Real;   // Fuerza a efectuar
      RESET : Bool;   // Salida de la maniobra
   END_VAR
   VAR_OUTPUT
      ACT : Bool;   // actuador de fuerza
   END_VAR
   VAR_IN_OUT
      bdfin_fuerza : Bool;   // señal que simboliza el final de al feurza aplicada
      Aviso_Error_Tiempo_Lim : Bool;
      Aviso_error_analogico : Bool;
      Fuerza_Real : Real;   // Valor de salida tratado por la funcion scale
   END_VAR
   VAR
      BDT : Bool;
      XMAN : Bool;
      Aviso_Interno_Tiempo : Bool;
      Aviso_Interno_Fin : Bool;
      Aviso_Interno_Error_Analógico : Bool;
   END_VAR
BEGIN

REGION Network 1: LLAMADAS INCONDICIONALES A BLOQUES

         CALL  "TRAT_SENSOR_FUERZA"
         ( RAW                    := #Fuerza_Bruta,
           BIPOLAR                := FALSE,
           HI_LIM                 := #HI_LIM,
           LO_LIM                 := #LO_LIM,
           FUERZA_NECESARIA       := #FUERZA_NECESARIA,
           RESET                  := #RESET,
           Aviso_Fuerza_Necesaria := #Aviso_Interno_Fin,
           Error                  := #Aviso_Interno_Error_Analógico,
           Real_Val               := #Fuerza_Real
         );
END_REGION

REGION Network 2: DESCONEXIÓN RESET
   // MAX PRIORITY
         A     #RESET;
         R     #BDT;

         R     #ACT;
         R     #Aviso_Error_Tiempo_Lim;
         R     #bdfin_fuerza;
         R     #Aviso_error_analogico;

         R     #Temp_Ciclo;
         FR    #Temp_Ciclo;

         BEC;
END_REGION

REGION Network 3: DESCONEXION ERROR TIEMPO LIMITE
         A     #Aviso_Interno_Tiempo;
         R     #BDT;

         S     #Aviso_Error_Tiempo_Lim;
         R     #Aviso_Interno_Tiempo;
         R     #Aviso_error_analogico;

         R     #Temp_Ciclo;
         FR    #Temp_Ciclo;
         R     #ACT;

         BEC;
END_REGION

REGION Network 4: DESCONEXION ERROR SEÑAL ANALÓGICA
         A     #Aviso_Interno_Error_Analógico;
         R     #BDT;
         S     #Aviso_error_analogico;
         R     #Aviso_Interno_Error_Analógico;
         R     #Aviso_Error_Tiempo_Lim;

         R     #Temp_Ciclo;
         FR    #Temp_Ciclo;
         R     #ACT;

         BEC;
END_REGION

REGION Network 5: DESCONEXION FIN MANIOBRA
         A     #Aviso_Interno_Fin;
         R     #BDT;
   //avisos externos
         S     #bdfin_fuerza;
         R     #Aviso_Interno_Fin;

         R     #Temp_Ciclo;
         FR    #Temp_Ciclo;
         R     #ACT;

         BEC;
END_REGION

REGION Network 6: CONEXION XMARCHA
         SET;

         L     #Tiempo_Max_Ciclo;
         SD    #Temp_Ciclo;

         FP    #BDT;
         S     #XMAN;
   //reseteo todos los avisos externos
         R     #bdfin_fuerza;
         R     #Aviso_error_analogico;
         R     #Aviso_Error_Tiempo_Lim;
END_REGION

REGION Network 7: TRAT ERROR TIEMPO
         A     #Temp_Ciclo;
         =     #Aviso_Interno_Tiempo;
END_REGION

REGION Network 8: ACTUADOR
         A     #XMAN;
         =     #ACT;
END_REGION
END_FUNCTION_BLOCK

FUNCTION_BLOCK "man_1A_ET_Reset"   // FB6, LAD
TITLE = Maniobra simple con gestión de error por tiempo límite
{ S7_Optimized_Access := 'TRUE' }
VERSION : 0.1
// Maniobra de una acción con error por tiempo limite
   VAR_INPUT
      SFIN : Bool;   // detector de finalización de maniobra
      tiempo_limite : S5Time := S5T#10s;   // tiempo máximo de duración
      T_limite : Timer;   // timer legacy
      RESET : Bool;   // entrada asíncrona, parada brusca de maniobra
   END_VAR
   VAR_OUTPUT
      ACT : Bool;   // actuador de maniobra
   END_VAR
   VAR_IN_OUT
      aviso_error_tiempo_limite : Bool;
      aviso_fin_maniobra : Bool;
   END_VAR
   VAR
      X_MAN : Bool;   // estado_maniobra_activa
      aviso_error_interno_tiempo_limite : Bool;
      aviso_interno_fin_maniobra : Bool;
      bit_de_trabajo : Bool;   // plantilla arranque
   END_VAR
BEGIN

REGION Network 1 (STL): DESCONEXION RESET (prioridad máxima)
   // primero mayor prioridad
   // borra todos los avisos (opcional)
   //evento asíncrono de parada brusca de maniobra
   //se pierde la unidad producida en el momento del RESET
   //al volver a entrar en producción, la ejecución de la maniobra comienza desde el principio
         A     #RESET;
         R     #bit_de_trabajo;
         R     #aviso_error_tiempo_limite;
         R     #aviso_fin_maniobra;
         R     #T_limite;
         FR    #T_limite;
         R     #ACT;
         BEC;
END_REGION

REGION Network 2 (STL): DESCONEXIÓN error tiempo limite
   // primero mayor prioridad
   //conectores de error- tiempo máximo de maniobra superado
         A     #aviso_error_interno_tiempo_limite;
         R     #bit_de_trabajo;
         S     #aviso_error_tiempo_limite;
         R     #aviso_error_interno_tiempo_limite;
         R     #T_limite;
         FR    #T_limite;
         R     #ACT;
         BEC;  //fin de ejecución de bloque
END_REGION

REGION Network 3 (STL): DESCONEXIÓN fin de maniobra
   // primero mayor prioridad
         A     #aviso_interno_fin_maniobra;
         R     #bit_de_trabajo;
         S     #aviso_fin_maniobra;
         R     #aviso_interno_fin_maniobra;
         R     #T_limite;  //necesario, el temporizador estará en uso
         FR    #T_limite;
         R     #ACT;
         BEC;
END_REGION

REGION Network 4 (STL): CONEXIÓN: activación de X_MAN (maniobra simple) y temporizador
   // Configuración de un  TON sin memoria como perro guardián
         SET;
   //configuración del temporizador: TON sin memoria como perro guardián
         L     #tiempo_limite;
         SD    #T_limite;
   //arranque
         FP    #bit_de_trabajo;
         S     #X_MAN;
   //reset todos los avisos externos
         R     #aviso_error_tiempo_limite;
         R     #aviso_fin_maniobra;
END_REGION

REGION Network 5: activación aviso de error por tiempo límite
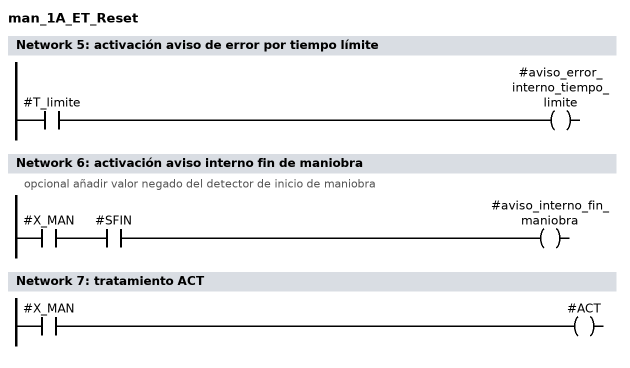
   RUNG wire#powerrail
      Contact( #T_limite )
      Coil( #aviso_error_interno_tiempo_limite )
   END_RUNG
   // the same network as SCL:
   #aviso_error_interno_tiempo_limite := #T_limite;
END_REGION

REGION Network 6: activación aviso interno fin de maniobra
   // opcional añadir valor negado del detector de inicio de maniobra
   RUNG wire#powerrail
      Contact( #X_MAN )
      Contact( #SFIN )
      Coil( #aviso_interno_fin_maniobra )
   END_RUNG
   // the same network as SCL:
   #aviso_interno_fin_maniobra := #X_MAN AND #SFIN;
END_REGION

REGION Network 7: tratamiento ACT
   RUNG wire#powerrail
      Contact( #X_MAN )
      Coil( #ACT )
   END_RUNG
   // the same network as SCL:
   #ACT := #X_MAN;
END_REGION
END_FUNCTION_BLOCK

FUNCTION_BLOCK "MOV_BRAZO_2"   // FB8, STL
{ S7_Optimized_Access := 'TRUE' }
VERSION : 0.1
// Maniobra para cuando el robot tiene que realizar una descarga en una maquina. Incluye  la carga y descarga de la pieza y la espera hasta que la máquina este descargada para poder introducir la pieza
   VAR_INPUT
      Sensor_Pieza : Bool;   // Sensor que detecta si hay una pieza que el robot tiene que coger
      Sensor_Pinza_Llena : Bool;   // Sensor que detecta si la pinza tiene una pieza o no
      Sensor_Llegada_a_Maquina : Bool;   // Sensor que detecta la llegada del robot a la máquina
      Sensor_Llegada_a_Buffer : Bool;   // Sensor que detecta que el robot ha llegado al buffer
      "Sensor_Llegada_a _Reposo" : Bool;   // Sensor que detecta la llegada del robot a la posición de reposo
      EMER : Bool;   // Entrada que indica la entrada del sistema en emergencia
      Tiempo_lim : S5Time;   // Tiempo limite de maniobra
      Timer_LIM : Timer;   // Temporizador para el tiempo limite de maniobra
   END_VAR
   VAR_OUTPUT
      MOV1 : Bool;   // Brazo se mueve a buffer
      MOV2 : Bool;   // Brazo se mueve a maquina
      MOV3 : Bool;   // Brazo se mueve a reposo
      ACT1 : Bool;   // Brazo coje pieza
      ACT2 : Bool;   // Brazo descarga pieza
   END_VAR
   VAR_IN_OUT
      Aviso_Error_Tiempo_Limite : Bool;   // Si se sobrepasa el tiempo se activa este aviso
      Aviso_Fin_Maniobra : Bool;   // Si la maniobra termina se activa este aviso para indicar que el brazo esta libre
      Aviso_Error_No_Pieza : Bool;   // Si no detecta una pieza cuando le han mandado a por una pieza el robot activa este error
      Aviso_Error_Pinza_Abierta : Bool;   // Si la pinza se abre en un momento que no deberia (MOV2 y WAIT1) se activa
   END_VAR
   VAR
      BDT : Bool;   // Bit de trabajo
      X1 : Bool;   // Etapa de MOV 1
      X2 : Bool;   // Etapa de ACT 1
      X3 : Bool;   // Etapa de MOV 2
      X4 : Bool;   // Etapa de WAIT 1
      X5 : Bool;   // Etapa de ACT2
      Aviso_Interno_Tiempo : Bool;
      Aviso_Interno_FIN : Bool;
      Aviso_Interno_Pinza_Abierta : Bool;
      Aviso_Interno_NO_Pieza : Bool;
   END_VAR
BEGIN

REGION Network 1: DESCONEXIÓN RESET
   // MAX PRIORITY
         A     #EMER;
         R     #BDT;
         R     #Aviso_Error_No_Pieza;
         R     #Aviso_Error_Pinza_Abierta;
         R     #Aviso_Error_Tiempo_Limite;
         R     #Aviso_Fin_Maniobra;
         R     #MOV1;
         R     #MOV2;
         R     #MOV3;
         R     #ACT1;
         R     #ACT2;

         R     #Timer_LIM;
         FR    #Timer_LIM;

         BEC;
END_REGION

REGION Network 2: DESCONEXION ERROR TIEMPO LIMITE
         A     #Aviso_Interno_Tiempo;
         R     #BDT;
         S     #Aviso_Error_Tiempo_Limite;
         R     #Aviso_Interno_Tiempo;
         R     #Timer_LIM;
         FR    #Timer_LIM;
         R     #MOV1;
         R     #MOV2;
         R     #MOV3;
         R     #ACT1;
         R     #ACT2;

         BEC;
END_REGION

REGION Network 3: DESCONEXION ERROR NO PIEZA
         A     #Aviso_Interno_NO_Pieza;
         R     #BDT;
         S     #Aviso_Error_No_Pieza;
         R     #Aviso_Interno_NO_Pieza;
         R     #Timer_LIM;
         FR    #Timer_LIM;
         R     #MOV1;
         R     #MOV2;
         R     #MOV3;
         R     #ACT1;
         R     #ACT2;

         BEC;
END_REGION

REGION Network 4: DESCONEXION ERROR PINZA ABIERTA
         A     #Aviso_Interno_Pinza_Abierta;
         R     #BDT;
         S     #Aviso_Error_Pinza_Abierta;
         R     #Aviso_Interno_Pinza_Abierta;
         R     #Timer_LIM;
         FR    #Timer_LIM;
         R     #MOV1;
         R     #MOV2;
         R     #MOV3;
         R     #ACT1;
         R     #ACT2;


         BEC;
END_REGION

REGION Network 5: DESCONEXION FIN MANIOBRA
         A     #Aviso_Interno_FIN;
         R     #BDT;
         S     #Aviso_Fin_Maniobra;
         R     #Aviso_Interno_FIN;
         R     #Timer_LIM;
         FR    #Timer_LIM;
         R     #MOV1;
         R     #MOV2;
         R     #MOV3;
         R     #ACT1;
         R     #ACT2;


         BEC;
END_REGION

REGION Network 6: CONEXION XMARCHA
         SET;
         L     #Tiempo_lim;
         SS    #Timer_LIM;
         FP    #BDT;

         S     #X1;
         R     #X2;
         R     #X3;
         R     #X4;
         R     #X5;
END_REGION

REGION Network 7: X1(Mov a maquina)->X2(captura de la pieza) //AÑADIR TEMPORIZADOR A T1
         A     #X1;
         A     #Sensor_Llegada_a_Maquina;  //sensor que indica he llegado a la maquina
         S     #X2;  //Estado que simboliza carga de la pieza
         R     #X1;
END_REGION

REGION Network 8: X2(captura de la pieza)->X3 (Mov a buffer con pieza)
         A     #X2;
         A     #Sensor_Pinza_Llena;  //tengo objeto
         S     #X3;  //Mov hacia buffer
         R     #X2;
END_REGION

REGION Network 9: X3(Mov a buffer con pieza)->X4(coloca pieza en buffer)
         A     #X3;
         A     #Sensor_Llegada_a_Buffer;  //llega al Buffer
         S     #X4;
         R     #X3;
END_REGION

REGION Network 10: X4 (coloca pieza en buffer ) -> X5(Mov a reposo)
         A     #X4;
         AN    #Sensor_Pinza_Llena;
         S     #X5;
         R     #X4;
END_REGION

REGION Network 11: X5(Mov a reposo)->FIN
         A     #X5;
         A     #"Sensor_Llegada_a _Reposo";
         S     #Aviso_Interno_FIN;
         R     #X5;
         R     #Timer_LIM;
         FR    #Timer_LIM;
END_REGION

REGION Network 12: TRAT X1
         A     #X1;
         AN    #Sensor_Pieza;
         S     #Aviso_Interno_NO_Pieza;  //Significa que va a por una pieza y de repente la pieza deja de estar.
   //Posible fallo de que el sensor no funcione o bien de pieza mal colocada, Requiere operario

         A     #X1;
         O;
         =     #MOV1;  //Indica que la máquina se mueve
END_REGION

REGION Network 13: TRAT X2
         A     #X2;
         =     #ACT1;
END_REGION

REGION Network 14: TRAT X3
         A     #X3;
         AN    #Sensor_Pinza_Llena;
         S     #Aviso_Interno_Pinza_Abierta;  //En el transporte la pinza de abre, la pieza se cae. ERROR GRAVE

         A     #X3;
         =     #MOV2;  //Indica que la máquina realiza el segundo movimiento
END_REGION

REGION Network 15: TRAT X4
         A     #X4;
         =     #ACT2;
END_REGION

REGION Network 16: TRAT X5
         A     #X5;
         =     #MOV3;
END_REGION

REGION Network 17: TRAT ERROR TIEMPO LIMITE
         A     #Timer_LIM;
         S     #Aviso_Error_Tiempo_Limite;
         R     #Timer_LIM;
         FR    #Timer_LIM;
END_REGION
END_FUNCTION_BLOCK

// folder: maquinas

FUNCTION_BLOCK "maq_temp"   // FB2, STL
TITLE = MAQUINA TEMPERATURA
{ S7_Optimized_Access := 'TRUE' }
VERSION : 0.1
// Trata la temperatura necesaria a la que debe trabajar la maquina, y da la señal de mando para que se ponga en funcionamiento la cinta y empezar el proceso
   VAR_INPUT
      START : Bool;
      REARME : Bool;
      EMER : Bool;
      Tiempo_MAX_maniobra : S5Time;   // timer de tiempo maximo de maniobra
      Tempo_maniobra : Timer;   // timer de tiempo por maniobra
      Temperatura_SENSOR : Int;   // Señal analógixa del sensor
      HI_LIM : Real;
      LO_LIM : Real;
      Modo_Foco : Bool;   // Selecciona el tipo de maquina. TRUE-Horno. FLASE-Tunel
      Aviso_Piezas_Cargadas : Bool;   // Se ha cargado el lote
      Aviso_Piezas_Descargadas : Bool;
      Temperatura_limite : Real;
      Temperatura_OK : Real;   // temperatura necesaria para que se inicie el procesado
   END_VAR
   VAR_OUTPUT
      FOCO : Bool;   // activa el foco correspondiente de la maquina
      MOV : Bool;
      Aviso_OK : Bool;
      Aviso_Standby : Bool;
   END_VAR
   VAR_IN_OUT
      Aviso_error_sincrono_EXT : Bool;
      Aviso_error_sensor_EXT : Bool;
      Temperatura_REAL : Real;   // Valor de salida tratado por la función scale
   END_VAR
   VAR
      BDT : Bool;
      OK : Bool;
      X_Standby : Bool;
      X_Espera : Bool;
      X_Mov : Bool;
      X_Foco : Bool;   // Espera a descarga antes de volver a standby
      X_EMER : Bool;
      X_error_SINC : Bool;
      X_error_SENSOR : Bool;
      Aviso_Tiempo_Lim_cinta : Bool;
      Aviso_Fin_Maniobra : Bool;
      Aviso_Error_Sensor : Bool;
      Mf_Piezas_cargadas : Bool;
      Mf_Piezas_descargadas : Bool;
      MOV_CINTA : "man_1A_ET_Reset";
   END_VAR
BEGIN

REGION Network 1: EMERGENCIA
   // Parada por evento asíncrono
         A     #EMER;
         S     #X_EMER;

   //ESTADOS
         R     #X_Standby;
         R     #X_Foco;
         R     #X_Espera;
         R     #X_Mov;
         R     #X_error_SINC;
         R     #X_error_SENSOR;

   //TEMPORIZADORES
         R     #Tempo_maniobra;
         FR    #Tempo_maniobra;
   //MANIOBRAS

         JCN   _EMER;

         CALL  "TRAT_SENSOR_TEMPERATURA"
         ( RAW                  := #Temperatura_SENSOR,
           BIPOLAR              := FALSE,
           HI_LIM               := #HI_LIM,
           LO_LIM               := #LO_LIM,
           Temperatura_limite   := #Temperatura_limite,
           Temperatura_OK       := #Temperatura_OK,
           Modo_FOCO            := #Modo_Foco,
           RESET                := TRUE,
           Aviso_Foco_encendido := #FOCO,
           Aviso_Foco_OK        := #OK,
           Error                := #Aviso_Error_Sensor,
           Real_Val             := "Temperatura_REAL_HORNO"
         );


         CALL  #MOV_CINTA
         ( SFIN                      := #Aviso_Piezas_Descargadas,
           tiempo_limite             := #Tiempo_MAX_maniobra,
           T_limite                  := #Tempo_maniobra,
           RESET                     := TRUE,
           ACT                       := #MOV,
           aviso_error_tiempo_limite := #Aviso_Tiempo_Lim_cinta,
           aviso_fin_maniobra        := #Aviso_Fin_Maniobra
         );

   _EMER:NOP   0;
END_REGION

REGION Network 2: Salida X_EMER a X_Standby
         A     #X_EMER;
         AN    #EMER;
         A     #REARME;
         S     #X_Standby;
         R     #X_EMER;
END_REGION

REGION Network 3: START===FALSE
         AN    #START;
         R     #BDT;

   //AVISOS
         R     #Aviso_error_sincrono_EXT;
         R     #Aviso_error_sensor_EXT;
         R     #Aviso_Tiempo_Lim_cinta;
         R     #Aviso_Error_Sensor;


   //TEMPORIZADORES
         R     #Tempo_maniobra;
         FR    #Tempo_maniobra;
   //MANIOBRAS

         JCN   _UNSTART;

         CALL  "TRAT_SENSOR_TEMPERATURA"
         ( RAW                  := #Temperatura_SENSOR,
           BIPOLAR              := FALSE,
           HI_LIM               := #HI_LIM,
           LO_LIM               := #LO_LIM,
           Temperatura_limite   := #Temperatura_limite,
           Temperatura_OK       := #Temperatura_OK,
           Modo_FOCO            := #Modo_Foco,
           RESET                := TRUE,
           Aviso_Foco_encendido := #FOCO,
           Aviso_Foco_OK        := #OK,
           Error                := #Aviso_Error_Sensor,
           Real_Val             := "Temperatura_REAL_HORNO"
         );

         CALL  #MOV_CINTA
         ( SFIN                      := #Aviso_Piezas_Descargadas,
           tiempo_limite             := #Tiempo_MAX_maniobra,
           T_limite                  := #Tempo_maniobra,
           RESET                     := TRUE,
           ACT                       := #MOV,
           aviso_error_tiempo_limite := #Aviso_Tiempo_Lim_cinta,
           aviso_fin_maniobra        := #Aviso_Fin_Maniobra
         );



   _UNSTART:NOP   0;

         AN    #START;
         BEC;
END_REGION

REGION Network 4: TRAT X_Error_SINC / X_Error_SENSOR
         O     #X_error_SINC;
         O     #X_error_SENSOR;
         R     #X_Foco;
         R     #X_Mov;

         JCN   _RESET_DE_ERROR;

   //TEMPORIZADOR
         R     #Tempo_maniobra;
         FR    #Tempo_maniobra;


         CALL  "TRAT_SENSOR_TEMPERATURA"
         ( RAW                  := #Temperatura_SENSOR,
           BIPOLAR              := FALSE,
           HI_LIM               := #HI_LIM,
           LO_LIM               := #LO_LIM,
           Temperatura_limite   := #Temperatura_limite,
           Temperatura_OK       := #Temperatura_OK,
           Modo_FOCO            := #Modo_Foco,
           RESET                := TRUE,
           Aviso_Foco_encendido := #FOCO,
           Aviso_Foco_OK        := #OK,
           Error                := #Aviso_Error_Sensor,
           Real_Val             := "Temperatura_REAL_HORNO"
         );


         CALL  #MOV_CINTA
         ( SFIN                      := #Aviso_Piezas_Descargadas,
           tiempo_limite             := #Tiempo_MAX_maniobra,
           T_limite                  := #Tempo_maniobra,
           RESET                     := TRUE,
           ACT                       := #MOV,
           aviso_error_tiempo_limite := #Aviso_Tiempo_Lim_cinta,
           aviso_fin_maniobra        := #Aviso_Fin_Maniobra
         );



   _RESET_DE_ERROR:NOP   0;
END_REGION

REGION Network 5: Salida X_ERROR_SINC a X_STANDBY
         A     #X_error_SINC;
         AN    #Aviso_error_sincrono_EXT;
         S     #X_Standby;
         R     #X_error_SINC;
END_REGION

REGION Network 6: Salida X_ERROR_SENSOR a X_STANDBY
         A     #X_error_SENSOR;
         AN    #Aviso_error_sensor_EXT;
         S     #X_Standby;
         R     #X_error_SENSOR;
END_REGION

REGION Network 7: START===TRUE
   // Conexión
         A     #START;
         FP    #BDT;

         R     #X_Espera;
         R     #X_Mov;
         R     #X_Foco;
         R     #X_error_SINC;
         R     #X_error_SENSOR;
         S     #X_Standby;
END_REGION

REGION Network 8: X_STANDBY ---> (X_FOCO + X_ESPERA) Divergencia
   // Activación por flanco
         A     #X_Standby;

         A(;
         A     #Aviso_Piezas_Cargadas;
         FP    #Mf_Piezas_cargadas;
         );

         R     #X_Standby;
         S     #X_Foco;
         S     #X_Espera;
END_REGION

REGION Network 9: X_ESPERA--->X_MOV
   // Subida con error por tiempo excedido
         A     #X_Espera;
         A     #OK;
         R     #X_Espera;
         S     #X_Mov;
END_REGION

REGION Network 10: ( X_FOCO + X_MOV ) ---> X_STANDBY Convergencia
         A     #X_Foco;
         A     #X_Mov;
         A(;
         A     #Aviso_Piezas_Descargadas;
         FP    #Mf_Piezas_descargadas;
         );

         R     #X_Foco;
         R     #X_Mov;
         S     #X_Standby;

   //TEMPORIZADORES
         R     #Tempo_maniobra;
         FR    #Tempo_maniobra;
   //ACTUADORES
         R     #FOCO;
         R     #MOV;
END_REGION

REGION Network 11: TRAT X_FOCO
         A     #X_Foco;
         JCN   _FOCO;

         CALL  "TRAT_SENSOR_TEMPERATURA"
         ( RAW                  := #Temperatura_SENSOR,
           BIPOLAR              := FALSE,
           HI_LIM               := #HI_LIM,
           LO_LIM               := #LO_LIM,
           Temperatura_limite   := #Temperatura_limite,
           Temperatura_OK       := #Temperatura_OK,
           Modo_FOCO            := #Modo_Foco,
           RESET                := FALSE,
           Aviso_Foco_encendido := #FOCO,
           Aviso_Foco_OK        := #OK,
           Error                := #Aviso_Error_Sensor,
           Real_Val             := #Temperatura_REAL
         );


   // salida por error (prioridad alta)
         A     #Aviso_Error_Sensor;
         R     #X_Mov;
         R     #X_Foco;
         S     #X_error_SENSOR;


   _FOCO:NOP   0;
END_REGION

REGION Network 12: TRAT X_MOV
         A     #OK;
         A     #X_Mov;

         JCN   _MOV_CINTA;

         CALL  #MOV_CINTA
         ( SFIN                      := #Aviso_Piezas_Descargadas,
           tiempo_limite             := #Tiempo_MAX_maniobra,
           T_limite                  := #Tempo_maniobra,
           RESET                     := FALSE,
           ACT                       := #MOV,
           aviso_error_tiempo_limite := #Aviso_Tiempo_Lim_cinta,
           aviso_fin_maniobra        := #Aviso_Fin_Maniobra
         );


   // salida por error (prioridad alta)
         A     #Aviso_Tiempo_Lim_cinta;
         R     #X_Mov;
         R     #X_Foco;
         S     #X_error_SINC;


   _MOV_CINTA:NOP   0;
END_REGION

REGION Network 13: Activación del aviso de error síncrono / error sensor / tempe OK
         A     #X_error_SINC;
         =     #Aviso_error_sincrono_EXT;
         A     #X_error_SENSOR;
         =     #Aviso_error_sensor_EXT;
         A     #OK;
         =     #Aviso_OK;
END_REGION

REGION Network 14: TRAT STANDBY
         A     #X_Standby;
         =     #Aviso_Standby;
END_REGION
END_FUNCTION_BLOCK

FUNCTION_BLOCK "PULIDORA"   // FB3, STL
TITLE = PULIDORA
{ S7_Optimized_Access := 'TRUE' }
VERSION : 0.1
// Encarga de realizar dos tipos de pulido sobre la pieza de llegada
   VAR_INPUT
      Spieza : Bool;   // llegada de una pieza a la maquina
      SFMovCab : Bool;   // sensor cabezal
      SFMovCab2 : Bool;   // sensor cabezal 2
      SF_Acercar : Bool;   // sensor de acercamiento
      SFPulido1 : Bool;   // sensor pulido
      SFPulido2 : Bool;   // sensor pulido 2
      SFCambio : Bool;   // senosr de cambio
      SFAlejar : Bool;   // senosr alejamiento
      SFGiro : Bool;   // sensor de giro
      SFGiro2 : Bool;   // sensor de giro 2
      T_Max_MovCab : S5Time;
      T_Max_Mov_Cab2 : S5Time;
      T_Max_Acercar : S5Time;
      T_Max_Pulido : S5Time;
      T_Max_Pulido2 : S5Time;
      T_Max_Cambio : S5Time;
      T_Max_Alejar : S5Time;
      T_Max_Giro : S5Time;
      T_Max_Giro2 : S5Time;
      TMovCab : Timer;
      TMovCab2 : Timer;
      TAcercar : Timer;
      TPulido1 : Timer;
      TPulido2 : Timer;
      TCambio : Timer;
      TAlejar : Timer;
      TGiro : Timer;
      TGiro2 : Timer;
      START : Bool;
      REARME : Bool;
      EMER : Bool;
   END_VAR
   VAR_OUTPUT
      Mover_Cabezal : Bool;
      Mover_Cabezal2 : Bool;
      Acercar_ : Bool;
      Pulido_ : Bool;
      Cambio_ : Bool;
      Pulido2_ : Bool;
      Alejar_ : Bool;
      Giro_ : Bool;
      Giro2 : Bool;
      Aviso_StandBy : Bool;
      Aviso_Error_Asíncrono : Bool;
   END_VAR
   VAR_IN_OUT
      Aviso_Error_Sincrono : Bool;
   END_VAR
   VAR
      MfError_Sincrono : Bool;
      MfSpieza : Bool;
      BdfMovCab : Bool;
      BdfMovCab2 : Bool;
      BdfAcercar : Bool;
      BdfPulido : Bool;
      BdfPulido2 : Bool;
      BdfCambio : Bool;
      BdfAlejar : Bool;
      BdfGiro : Bool;
      BdfGiro2 : Bool;
      Bit_De_Trabajo : Bool;
      Aviso_Error_MovCab : Bool;
      Aviso_Error_MovCab2 : Bool;
      Aviso_Error_Acercar : Bool;
      Aviso_Error_Pulido : Bool;
      Aviso_Error_Cambio : Bool;
      Aviso_Error_Pulido2 : Bool;
      Aviso_Error_Alejar : Bool;
      Aviso_Error_Giro : Bool;
      Aviso_Error_Giro2 : Bool;
      man_Mov_Cab : "man_1A_ET_Reset";
      man_Mov_Cab2 : "man_1A_ET_Reset";
      man_Acercar : "man_1A_ET_Reset";
      man_Pulido : "man_1A_ET_Reset";
      man_Cambio : "man_1A_ET_Reset";
      man_Pulido2 : "man_1A_ET_Reset";
      man_Alejar : "man_1A_ET_Reset";
      man_Giro : "man_1A_ET_Reset";
      man_Giro2 : "man_1A_ET_Reset";
      X0_Stdby : Bool;
      X1_Espero_Giro_Hacia_Brazo : Bool;
      X_Girar_hacia_Pulidora : Bool;
      X_Girar_hacia_Brazo : Bool;
      X_Acercar_Pulidora : Bool;
      X_Pulir1 : Bool;
      X_Pulir2 : Bool;
      X_Cambio : Bool;
      X_Alejar_Pulidora : Bool;
      X_Mov_Cab_Con_Pulidora : Bool;
      X_Mov_Cab_Con_pulidora2 : Bool;
      X_EMER : Bool;
      X_error_sincrono : Bool;
   END_VAR
BEGIN

REGION Network 1: EMERGENCIA
         A     #EMER;
         S     #X_EMER;
         S     #Aviso_Error_Asíncrono;
         R     #X0_Stdby;
         R     #X1_Espero_Giro_Hacia_Brazo;
         R     #X_Acercar_Pulidora;
         R     #X_Alejar_Pulidora;
         R     #X_Cambio;
         R     #X_error_sincrono;
         R     #Aviso_Error_Sincrono;
         R     #X_Mov_Cab_Con_Pulidora;
         R     #X_Mov_Cab_Con_pulidora2;
         R     #X_Girar_hacia_Brazo;
         R     #X_Pulir1;
         R     #X_Pulir2;

         JCN   _aviso_emergencia;
         CALL  #man_Acercar
         ( SFIN                      := ,
           tiempo_limite             := ,
           T_limite                  := #TAcercar,
           RESET                     := TRUE,
           ACT                       := #Acercar_,
           aviso_error_tiempo_limite := #Aviso_Error_Acercar,
           aviso_fin_maniobra        := #BdfAcercar
         );
         CALL  #man_Alejar
         ( SFIN                      := ,
           tiempo_limite             := ,
           T_limite                  := #TAlejar,
           RESET                     := TRUE,
           ACT                       := #Alejar_,
           aviso_error_tiempo_limite := #Aviso_Error_Alejar,
           aviso_fin_maniobra        := #BdfAlejar
         );
         CALL  #man_Cambio
         ( SFIN                      := ,
           tiempo_limite             := ,
           T_limite                  := #TCambio,
           RESET                     := TRUE,
           ACT                       := #Cambio_,
           aviso_error_tiempo_limite := #Aviso_Error_Cambio,
           aviso_fin_maniobra        := #BdfCambio
         );
         CALL  #man_Giro
         ( SFIN                      := ,
           tiempo_limite             := ,
           T_limite                  := #TGiro,
           RESET                     := TRUE,
           ACT                       := #Giro_,
           aviso_error_tiempo_limite := #Aviso_Error_Giro,
           aviso_fin_maniobra        := #BdfGiro
         );
         CALL  #man_Giro2
         ( SFIN                      := ,
           tiempo_limite             := ,
           T_limite                  := #TGiro2,
           RESET                     := TRUE,
           ACT                       := #Giro2,
           aviso_error_tiempo_limite := #Aviso_Error_Giro2,
           aviso_fin_maniobra        := #BdfGiro2
         );
         CALL  #man_Mov_Cab
         ( SFIN                      := #SFMovCab,
           tiempo_limite             := #T_Max_MovCab,
           T_limite                  := #TMovCab,
           RESET                     := TRUE,
           ACT                       := #Mover_Cabezal,
           aviso_error_tiempo_limite := #Aviso_Error_MovCab,
           aviso_fin_maniobra        := #BdfMovCab
         );
         CALL  #man_Mov_Cab2
         ( SFIN                      := ,
           tiempo_limite             := ,
           T_limite                  := #TMovCab2,
           RESET                     := TRUE,
           ACT                       := #Mover_Cabezal2,
           aviso_error_tiempo_limite := #Aviso_Error_MovCab2,
           aviso_fin_maniobra        := #BdfMovCab2
         );
         CALL  #man_Pulido
         ( SFIN                      := ,
           tiempo_limite             := ,
           T_limite                  := #TPulido1,
           RESET                     := TRUE,
           ACT                       := #Pulido_,
           aviso_error_tiempo_limite := #Aviso_Error_Pulido,
           aviso_fin_maniobra        := #BdfPulido
         );
         CALL  #man_Pulido2
         ( SFIN                      := ,
           tiempo_limite             := ,
           T_limite                  := #TPulido2,
           RESET                     := TRUE,
           ACT                       := #Pulido2_,
           aviso_error_tiempo_limite := #Aviso_Error_Pulido2,
           aviso_fin_maniobra        := #BdfPulido2
         );
   _aviso_emergencia:NOP   0;
END_REGION

REGION Network 2: REARME
         A     #X_EMER;
         AN    #EMER;
         A     #REARME;
         S     #X0_Stdby;
         R     #X_EMER;
         R     #Aviso_Error_Asíncrono;
END_REGION

REGION Network 3: Error_Por_Evento_síncrono
         A     #X_error_sincrono;
         R     #X0_Stdby;
         R     #X1_Espero_Giro_Hacia_Brazo;
         R     #X_Acercar_Pulidora;
         R     #X_Alejar_Pulidora;
         R     #X_Cambio;
         R     #X_Girar_hacia_Brazo;
         R     #X_Girar_hacia_Pulidora;
         R     #X_Mov_Cab_Con_Pulidora;
         R     #X_Mov_Cab_Con_pulidora2;
         R     #X_Pulir1;
         R     #X_Pulir2;
   // mfErrorSincrono
         FP    #MfError_Sincrono;
         S     #Aviso_Error_Sincrono;
END_REGION

REGION Network 4: Vuelta StdBy despues de errores sincronos
         A     #X_error_sincrono;
         AN    #Aviso_Error_Sincrono;
         S     #X0_Stdby;
         R     #X_error_sincrono;
END_REGION

REGION Network 5: START=TRUE
         A     #START;
         SET;
         FP    #Bit_De_Trabajo;
         S     #X0_Stdby;
         R     #X_EMER;
         R     #X_error_sincrono;
         R     #X1_Espero_Giro_Hacia_Brazo;
         R     #X_Acercar_Pulidora;
         R     #X_Alejar_Pulidora;
         R     #X_Cambio;
         R     #X_Girar_hacia_Brazo;
         R     #X_Girar_hacia_Pulidora;
         R     #X_Mov_Cab_Con_Pulidora;
         R     #X_Mov_Cab_Con_pulidora2;
         R     #X_Pulir1;
         R     #X_Pulir2;
END_REGION

REGION Network 6: START=FALSE
         AN    #START;
         R     #Bit_De_Trabajo;
         R     #Aviso_Error_Sincrono;
         R     #Aviso_StandBy;
         R     #Aviso_Error_Asíncrono;

         JCN   _Reset;
         CALL  #man_Acercar
         ( SFIN                      := ,
           tiempo_limite             := ,
           T_limite                  := ,
           RESET                     := TRUE,
           ACT                       := #Acercar_,
           aviso_error_tiempo_limite := #Aviso_Error_Acercar,
           aviso_fin_maniobra        := #BdfAcercar
         );
         CALL  #man_Alejar
         ( SFIN                      := ,
           tiempo_limite             := ,
           T_limite                  := ,
           RESET                     := TRUE,
           ACT                       := #Alejar_,
           aviso_error_tiempo_limite := #Aviso_Error_Alejar,
           aviso_fin_maniobra        := #BdfAlejar
         );
         CALL  #man_Cambio
         ( SFIN                      := ,
           tiempo_limite             := ,
           T_limite                  := ,
           RESET                     := TRUE,
           ACT                       := #Cambio_,
           aviso_error_tiempo_limite := #Aviso_Error_Cambio,
           aviso_fin_maniobra        := #BdfCambio
         );
         CALL  #man_Giro
         ( SFIN                      := ,
           tiempo_limite             := ,
           T_limite                  := ,
           RESET                     := TRUE,
           ACT                       := #Giro_,
           aviso_error_tiempo_limite := #Aviso_Error_Giro,
           aviso_fin_maniobra        := #BdfGiro
         );
         CALL  #man_Giro2
         ( SFIN                      := ,
           tiempo_limite             := ,
           T_limite                  := ,
           RESET                     := TRUE,
           ACT                       := #Giro2,
           aviso_error_tiempo_limite := #Aviso_Error_Giro2,
           aviso_fin_maniobra        := #BdfGiro2
         );
         CALL  #man_Mov_Cab
         ( SFIN                      := ,
           tiempo_limite             := ,
           T_limite                  := ,
           RESET                     := TRUE,
           ACT                       := #Mover_Cabezal,
           aviso_error_tiempo_limite := #Aviso_Error_MovCab,
           aviso_fin_maniobra        := #BdfMovCab
         );
         CALL  #man_Mov_Cab2
         ( SFIN                      := ,
           tiempo_limite             := ,
           T_limite                  := ,
           RESET                     := TRUE,
           ACT                       := #Mover_Cabezal2,
           aviso_error_tiempo_limite := #Aviso_Error_MovCab2,
           aviso_fin_maniobra        := #BdfMovCab2
         );
         CALL  #man_Pulido
         ( SFIN                      := ,
           tiempo_limite             := ,
           T_limite                  := ,
           RESET                     := TRUE,
           ACT                       := #Pulido_,
           aviso_error_tiempo_limite := #Aviso_Error_Pulido,
           aviso_fin_maniobra        := #BdfPulido
         );
         CALL  #man_Pulido2
         ( SFIN                      := ,
           tiempo_limite             := ,
           T_limite                  := ,
           RESET                     := TRUE,
           ACT                       := #Pulido2_,
           aviso_error_tiempo_limite := #Aviso_Error_Pulido2,
           aviso_fin_maniobra        := #BdfPulido2
         );
   _Reset:NOP   0;
END_REGION

REGION Network 7: X0->X_Giro_Hacia_Pulidora,X2,X3
         A     #X0_Stdby;
         A(;
         A     #Spieza;
         FP    #MfSpieza;
         );
         R     #X0_Stdby;
         S     #X_Girar_hacia_Pulidora;
END_REGION

REGION Network 8: X_Giro_Hacia_Pulidora(Soporte)->XAcercar_Pulidora
         A     #X_Girar_hacia_Pulidora;
         JCN   _Llamada_man_giro_HaciaPulidora;
         CALL  #man_Giro
         ( SFIN                      := #SFGiro,
           tiempo_limite             := #T_Max_Giro,
           T_limite                  := #TGiro,
           RESET                     := FALSE,
           ACT                       := #Giro_,
           aviso_error_tiempo_limite := #Aviso_Error_Giro,
           aviso_fin_maniobra        := #BdfGiro
         );
         A     #Aviso_Error_Giro;
         R     #X_Girar_hacia_Pulidora;
         S     #X_error_sincrono;

         A     #BdfGiro;
         R     #X_Girar_hacia_Pulidora;
         S     #X_Acercar_Pulidora;

   _Llamada_man_giro_HaciaPulidora:NOP   0;
END_REGION

REGION Network 9: X_Acercar_Pulidora->X_Pulir,Mover_Con_Pulidora(Cabezal)
         A     #X_Acercar_Pulidora;
         JCN   _Llamada_man_Acercar_Pulidora;
         CALL  #man_Acercar
         ( SFIN                      := #SF_Acercar,
           tiempo_limite             := #T_Max_Acercar,
           T_limite                  := #TAcercar,
           RESET                     := FALSE,
           ACT                       := #Acercar_,
           aviso_error_tiempo_limite := #Aviso_Error_Acercar,
           aviso_fin_maniobra        := #BdfAcercar
         );
         A     #Aviso_Error_Acercar;
         R     #X_Acercar_Pulidora;
         S     #X_error_sincrono;


         A     #BdfAcercar;
         R     #X_Acercar_Pulidora;
         S     #X_Pulir1;
         S     #X_Mov_Cab_Con_Pulidora;

   _Llamada_man_Acercar_Pulidora:NOP   0;
END_REGION

REGION Network 10: X_Pulir,Mov_Cab_Con_Pulidora->X_Cambio
         A     #X_Pulir1;
         A     #X_Mov_Cab_Con_Pulidora;
         JCN   _Llamada_man_Pulir1_y_Mov_Cabezal;
         CALL  #man_Pulido
         ( SFIN                      := #SFPulido1,
           tiempo_limite             := #T_Max_Pulido,
           T_limite                  := #TPulido1,
           RESET                     := FALSE,
           ACT                       := #Pulido_,
           aviso_error_tiempo_limite := #Aviso_Error_Pulido,
           aviso_fin_maniobra        := #BdfPulido
         );

         CALL  #man_Mov_Cab
         ( SFIN                      := #SFMovCab,
           tiempo_limite             := #T_Max_MovCab,
           T_limite                  := #TMovCab,
           RESET                     := FALSE,
           ACT                       := #Mover_Cabezal,
           aviso_error_tiempo_limite := #Aviso_Error_MovCab,
           aviso_fin_maniobra        := #BdfMovCab
         );
   // Error Por tiempo de maniobra
         A(;
         O     #Aviso_Error_Pulido;
         O     #Aviso_Error_MovCab;
         );
         R     #X_Pulir1;
         R     #Mover_Cabezal;
         S     #X_error_sincrono;
   // Paso de una maniobra a otra
         A     #BdfPulido;
         A     #BdfMovCab;
         R     #Mover_Cabezal;
         R     #X_Pulir1;
         S     #X_Cambio;
   _Llamada_man_Pulir1_y_Mov_Cabezal:NOP   0;
END_REGION

REGION Network 11: X_Cambio->X_Pulir2, X_MovCab2
         A     #X_Cambio;
         JCN   _LLamada_man_Cambio;
         CALL  #man_Cambio
         ( SFIN                      := #SFCambio,
           tiempo_limite             := #T_Max_Cambio,
           T_limite                  := #TCambio,
           RESET                     := FALSE,
           ACT                       := #Cambio_,
           aviso_error_tiempo_limite := #Aviso_Error_Cambio,
           aviso_fin_maniobra        := #BdfCambio
         );
         A     #Aviso_Error_Cambio;
         R     #X_Cambio;
         S     #X_error_sincrono;

         A     #BdfCambio;
         R     #X_Cambio;
         S     #X_Pulir2;
         S     #X_Mov_Cab_Con_pulidora2;

   _LLamada_man_Cambio:NOP   0;
END_REGION

REGION Network 12: X_Pulir 2,X_Mov_Cab_Con_pulidora-> Alejar_Pulidora
         A     #X_Pulir2;
         A     #X_Mov_Cab_Con_pulidora2;
         JCN   _Llamada_man_Pulir2;
         CALL  #man_Pulido2
         ( SFIN                      := #SFPulido2,
           tiempo_limite             := #T_Max_Pulido2,
           T_limite                  := #TPulido2,
           RESET                     := FALSE,
           ACT                       := #Pulido2_,
           aviso_error_tiempo_limite := #Aviso_Error_Pulido2,
           aviso_fin_maniobra        := #BdfPulido2
         );
         CALL  #man_Mov_Cab2
         ( SFIN                      := #SFMovCab2,
           tiempo_limite             := #T_Max_Mov_Cab2,
           T_limite                  := #TMovCab2,
           RESET                     := FALSE,
           ACT                       := #Mover_Cabezal2,
           aviso_error_tiempo_limite := #Aviso_Error_MovCab2,
           aviso_fin_maniobra        := #BdfMovCab2
         );



         A(;
         O     #Aviso_Error_Pulido2;
         O     #Aviso_Error_MovCab2;
         );
         R     #X_Pulir2;
         R     #Mover_Cabezal2;
         S     #X_error_sincrono;
   // PAso de una maniobra a otra
         A     #BdfPulido2;
         A     #BdfMovCab2;
         R     #Mover_Cabezal2;
         R     #X_Pulir2;
         S     #X_Alejar_Pulidora;

   _Llamada_man_Pulir2:NOP   0;
END_REGION

REGION Network 13: X_Alejar_Pulidora->X_Giro_Hacia_Brazo
         A     #X_Alejar_Pulidora;
         JCN   _Llamada_man_Alejar_Pulidora;
         CALL  #man_Alejar
         ( SFIN                      := #SFAlejar,
           tiempo_limite             := #T_Max_Alejar,
           T_limite                  := #TAlejar,
           RESET                     := FALSE,
           ACT                       := #Alejar_,
           aviso_error_tiempo_limite := #Aviso_Error_Alejar,
           aviso_fin_maniobra        := #BdfAlejar
         );
         A     #Aviso_Error_Alejar;
         R     #X_Alejar_Pulidora;
         S     #X_error_sincrono;

         A     #BdfAlejar;
         R     #X_Alejar_Pulidora;
         S     #X_Girar_hacia_Brazo;

   _Llamada_man_Alejar_Pulidora:NOP   0;
END_REGION

REGION Network 14: X_Giro_Hacia_Brazo->X2_Espero_Brazo
         A     #X_Girar_hacia_Brazo;
         JCN   _Llamada_man_giro_HaciaBrazo;
         CALL  #man_Giro2
         ( SFIN                      := #SFGiro2,
           tiempo_limite             := #T_Max_Giro2,
           T_limite                  := #TGiro2,
           RESET                     := FALSE,
           ACT                       := #Giro2,
           aviso_error_tiempo_limite := #Aviso_Error_Giro2,
           aviso_fin_maniobra        := #BdfGiro2
         );
         A     #Aviso_Error_Giro2;
         R     #X_Girar_hacia_Brazo;
         S     #X_error_sincrono;

         A     #BdfGiro2;
         R     #X_Girar_hacia_Brazo;
         S     #X1_Espero_Giro_Hacia_Brazo;
   _Llamada_man_giro_HaciaBrazo:NOP   0;
END_REGION

REGION Network 15: X1_EsperoBrazo->X0_StdBy
         A     #X1_Espero_Giro_Hacia_Brazo;
         AN    #Spieza;
         R     #X1_Espero_Giro_Hacia_Brazo;
         S     #X0_Stdby;
END_REGION

REGION Network 16: Aviso Stdby
         A     #X0_Stdby;
         =     #Aviso_StandBy;
END_REGION
END_FUNCTION_BLOCK

FUNCTION_BLOCK "CONFORMADORA"   // FB5, STL
TITLE = COMFORMADORA
{ S7_Optimized_Access := 'TRUE' }
VERSION : 0.1
// Realiza una fuerza hasta llegar al humbral requerido. Tratamiento de señal analógica
   VAR_INPUT
      START : Bool;
      REARME : Bool;
      EMER : Bool;
      S_fin : Bool;   // Señaliza la llegada del piston de la maquina a su posicion inicial
      Tiempo_MAX_maniobra : S5Time;
      Temp_Ciclo_compre : Timer;   // timer de la compresion
      Temp_Ciclo_descompre : Timer;   // timer de la descompresion
      Fuerza_SENSOR : Int;   // Señal analogica que recibe el sensor
      HI_LIM : Real;
      LO_LIM : Real;
      Aviso_Pieza_Cargada : Bool;   // Se ha cargado el lote en la conformadora
      Aviso_Pieza_Descargada : Bool;   // Se ha descargado el lote en la conformadora
      FUERZA_NECESARIA : Real;
   END_VAR
   VAR_OUTPUT
      COMPRIMIR : Bool;
      DESCOMPRIR : Bool;
      Aviso_Standby : Bool;   // Aviso del estado de Standby
   END_VAR
   VAR_IN_OUT
      Aviso_error_sincrono_EXT : Bool;
      Aviso_error_sensor_EXT : Bool;
      FUERZA_REAL : Real;   // Valor de salida tratado por la función scale
   END_VAR
   VAR
      BDT : Bool;
      X_Standby : Bool;
      X_Conprimiendo : Bool;
      X_Descomprimiendo : Bool;
      X_Espera : Bool;   // Espera a descarga antes de volver a standby
      X_EMER : Bool;
      X_error_SINC : Bool;   // error sincrono
      X_error_SENSOR : Bool;   // errror asincrono
      Aviso_Tiempo_Lim_descompre : Bool;
      Aviso_Tiempo_Lim_compre : Bool;
      Aviso_Fin_Compresion : Bool;
      Aviso_Fin_Descompresion : Bool;
      Aviso_Error_Sensor : Bool;
      Mf_Pieza_cargada : Bool;
      MOV_COMPRIMIR : "MOV_CONFOR_FUERZA";
      MOV_DESCOMPRIMIR : "man_1A_ET_Reset";
   END_VAR
BEGIN

REGION Network 1: EMERGENCIA
   // Parada por evento asíncrono
         A     #EMER;
         S     #X_EMER;

   //ESTADOS
         R     #X_Conprimiendo;
         R     #X_Espera;
         R     #X_Standby;
         R     #X_Descomprimiendo;
         R     #X_error_SINC;
         R     #X_error_SENSOR;

   //TEMPORIZADORES
         R     #Temp_Ciclo_descompre;
         FR    #Temp_Ciclo_descompre;
   //MANIOBRAS

         JCN   _EMER;

         CALL  #MOV_COMPRIMIR
         ( Tiempo_Max_Ciclo       := #Tiempo_MAX_maniobra,
           Temp_Ciclo             := #Temp_Ciclo_compre,
           Fuerza_Bruta           := #Fuerza_SENSOR,
           HI_LIM                 := #HI_LIM,
           LO_LIM                 := #LO_LIM,
           FUERZA_NECESARIA       := #FUERZA_NECESARIA,
           RESET                  := TRUE,
           ACT                    := #COMPRIMIR,
           bdfin_fuerza           := #Aviso_Fin_Compresion,
           Aviso_Error_Tiempo_Lim := #Aviso_Tiempo_Lim_compre,
           Aviso_error_analogico  := #Aviso_Error_Sensor,
           Fuerza_Real            := #FUERZA_REAL
         );

         CALL  #MOV_DESCOMPRIMIR
         ( SFIN                      := #S_fin,
           tiempo_limite             := #Tiempo_MAX_maniobra,
           T_limite                  := #Temp_Ciclo_descompre,
           RESET                     := TRUE,
           ACT                       := #DESCOMPRIR,
           aviso_error_tiempo_limite := #Aviso_Tiempo_Lim_descompre,
           aviso_fin_maniobra        := #Aviso_Fin_Descompresion
         );



   _EMER:NOP   0;
END_REGION

REGION Network 2: SALIDA DE X_EMER a X_STANDBY
         A     #X_EMER;
         AN    #EMER;
         A     #REARME;
         S     #X_Standby;
         R     #X_EMER;
END_REGION

REGION Network 3: START===FALSE
         AN    #START;
         R     #BDT;

   //AVISOS
         R     #Aviso_error_sincrono_EXT;
         R     #Aviso_Standby;
         R     #Aviso_Tiempo_Lim_descompre;
   //TEMPORIZADORES
         R     #Temp_Ciclo_descompre;
         FR    #Temp_Ciclo_descompre;
   //MANIOBRAS

         JCN   _UNSTART;

         CALL  #MOV_COMPRIMIR
         ( Tiempo_Max_Ciclo       := #Tiempo_MAX_maniobra,
           Temp_Ciclo             := #Temp_Ciclo_compre,
           Fuerza_Bruta           := #Fuerza_SENSOR,
           HI_LIM                 := #HI_LIM,
           LO_LIM                 := #LO_LIM,
           FUERZA_NECESARIA       := #FUERZA_NECESARIA,
           RESET                  := TRUE,
           ACT                    := #COMPRIMIR,
           bdfin_fuerza           := #Aviso_Fin_Compresion,
           Aviso_Error_Tiempo_Lim := #Aviso_Tiempo_Lim_compre,
           Aviso_error_analogico  := #Aviso_Error_Sensor,
           Fuerza_Real            := #FUERZA_REAL
         );

         CALL  #MOV_DESCOMPRIMIR
         ( SFIN                      := #S_fin,
           tiempo_limite             := #Tiempo_MAX_maniobra,
           T_limite                  := #Temp_Ciclo_descompre,
           RESET                     := TRUE,
           ACT                       := #DESCOMPRIR,
           aviso_error_tiempo_limite := #Aviso_Tiempo_Lim_descompre,
           aviso_fin_maniobra        := #Aviso_Fin_Descompresion
         );

   _UNSTART:NOP   0;

         AN    #START;
         BEC;
END_REGION

REGION Network 4: TRAT X_Error_SINC / X_Error_SENSOR
         O     #X_error_SINC;
         O     #X_error_SENSOR;
         R     #X_Conprimiendo;
         R     #X_Descomprimiendo;

         JCN   _RESET_DE_ERROR;

         CALL  #MOV_COMPRIMIR
         ( Tiempo_Max_Ciclo       := #Tiempo_MAX_maniobra,
           Temp_Ciclo             := #Temp_Ciclo_compre,
           Fuerza_Bruta           := #Fuerza_SENSOR,
           HI_LIM                 := #HI_LIM,
           LO_LIM                 := #LO_LIM,
           FUERZA_NECESARIA       := #FUERZA_NECESARIA,
           RESET                  := TRUE,
           ACT                    := #COMPRIMIR,
           bdfin_fuerza           := #Aviso_Fin_Compresion,
           Aviso_Error_Tiempo_Lim := #Aviso_Tiempo_Lim_compre,
           Aviso_error_analogico  := #Aviso_Error_Sensor,
           Fuerza_Real            := #FUERZA_REAL
         );

         CALL  #MOV_DESCOMPRIMIR
         ( SFIN                      := #S_fin,
           tiempo_limite             := #Tiempo_MAX_maniobra,
           T_limite                  := #Temp_Ciclo_descompre,
           RESET                     := TRUE,
           ACT                       := #DESCOMPRIR,
           aviso_error_tiempo_limite := #Aviso_Tiempo_Lim_descompre,
           aviso_fin_maniobra        := #Aviso_Fin_Descompresion
         );

   _RESET_DE_ERROR:NOP   0;
END_REGION

REGION Network 5: SALIDA X_ERROR_SINC / X_ERROR_SENSOR a X_STANDBY
         A     #X_error_SINC;
         AN    #Aviso_error_sincrono_EXT;
         S     #X_Standby;
         R     #X_error_SINC;

         A     #X_error_SENSOR;
         AN    #Aviso_error_sensor_EXT;
         S     #X_Standby;
         R     #X_error_SENSOR;
END_REGION

REGION Network 6: START===TRUE
   // Conexión
         A     #START;
         FP    #BDT;

         S     #X_Standby;
         R     #X_Conprimiendo;
         R     #X_Descomprimiendo;
         R     #X_Espera;
         R     #X_error_SINC;
END_REGION

REGION Network 7: X_STANDBY--->X__COMPRIMIENDO
   // Activación por flanco
         A     #X_Standby;

         A(;
         A     #Aviso_Pieza_Cargada;
         FP    #Mf_Pieza_cargada;
         );

         S     #X_Conprimiendo;
         R     #X_Standby;
END_REGION

REGION Network 8: TRAT X__COMPRIMIENDO
         A     #X_Conprimiendo;

         JCN   _COMPRIMIENDO;

         CALL  #MOV_COMPRIMIR
         ( Tiempo_Max_Ciclo       := #Tiempo_MAX_maniobra,
           Temp_Ciclo             := #Temp_Ciclo_compre,
           Fuerza_Bruta           := #Fuerza_SENSOR,
           HI_LIM                 := #HI_LIM,
           LO_LIM                 := #LO_LIM,
           FUERZA_NECESARIA       := #FUERZA_NECESARIA,
           RESET                  := FALSE,
           ACT                    := #COMPRIMIR,
           bdfin_fuerza           := #Aviso_Fin_Compresion,
           Aviso_Error_Tiempo_Lim := #Aviso_Tiempo_Lim_compre,
           Aviso_error_analogico  := #Aviso_Error_Sensor,
           Fuerza_Real            := #FUERZA_REAL
         );


         A     #Aviso_Fin_Compresion;
         S     #X_Descomprimiendo;
         R     #X_Conprimiendo;

         A     #Aviso_Tiempo_Lim_compre;
         S     #X_error_SINC;
         R     #X_Conprimiendo;

         A     #Aviso_Error_Sensor;
         S     #X_error_SENSOR;
         R     #X_Conprimiendo;


   _COMPRIMIENDO:NOP   0;
END_REGION

REGION Network 9: TRAT X_DESCOMPRIMIENDO
   // Subida con error por tiempo excedido
         A     #X_Descomprimiendo;

         JCN   _DESCOMPRIMIENDO;

         CALL  #MOV_DESCOMPRIMIR
         ( SFIN                      := #S_fin,
           tiempo_limite             := #Tiempo_MAX_maniobra,
           T_limite                  := #Temp_Ciclo_descompre,
           RESET                     := FALSE,
           ACT                       := #DESCOMPRIR,
           aviso_error_tiempo_limite := #Aviso_Tiempo_Lim_descompre,
           aviso_fin_maniobra        := #Aviso_Fin_Descompresion
         );


         A     #Aviso_Fin_Descompresion;
         S     #X_Espera;
         R     #X_Descomprimiendo;

         A     #Aviso_Tiempo_Lim_descompre;
         S     #X_error_SINC;
         R     #X_Conprimiendo;


   _DESCOMPRIMIENDO:NOP   0;
END_REGION

REGION Network 10: X_ESPERA--->X_STANDBY
         A     #X_Espera;
         A     #Aviso_Pieza_Descargada;
         S     #X_Standby;
         R     #X_Espera;
END_REGION

REGION Network 11: Activación del aviso de error síncrono
   // Segmento de prioridad
         A     #X_error_SINC;
         =     #Aviso_error_sincrono_EXT;
         A     #X_error_SENSOR;
         =     #Aviso_error_sensor_EXT;
END_REGION

REGION Network 12: TRAT X_STANDBY
         A     #X_Standby;
         =     #Aviso_Standby;
END_REGION
END_FUNCTION_BLOCK

FUNCTION_BLOCK "ROBOT"   // FB7, STL
TITLE = BRAZO ROBOT
{ S7_Optimized_Access := 'TRUE' }
VERSION : 0.1
// Maniobra 1
// Parte de una posicion inicial,  coge una pieza y  la deposita en otro apartado siempre y cuando la maquina en cuestion esté disponible, vuelve a su posición inicial.
// Maniobra 2
// Parte de una posicion inicial,  coge una pieza y  la deposita en otro apartado, vuelve a su posición inicial.
// 
// Error por tiempo limite.
// Erro por pinza.
   VAR_INPUT
      Sensor_Pieza : Bool;   // Sensor que detecta si hay una pieza que el robot tiene que cojer
      Sensor_Pinza_Llena : Bool;   // Sensor que detecta si la pinza tiene una pieza o no
      Sensor_Llegada_Carga : Bool;   // Sensor que detecta si el robot ha llegado al buffer de entrada
      Sensor_Llegada_Descarga : Bool;   // Sensor que detecta si el robot ha llegado a la salida de la maquina
      Sensor_Llegada_a_Reposo : Bool;   // Sensor que detecta si el robot ha llegado a estado de reposo
      START : Bool;   // Entrada que indica al robot que esta encendido
      EMER : Bool;   // Entrada que indica emergencia
      REARME : Bool;   // Entrada para rearmar el robot en caso de emergencia
      Tiempo_lim : S5Time;   // Tiempo limite de operación del robot
      Timer_LIM : Timer;   // Temporizador para el tiempo limite
      X_Marcha_1 : Bool;   // Modo de marcha 1
      X_Marcha_2 : Bool;   // Modo de marcha 2
   END_VAR
   VAR_OUTPUT
      Mov1 : Bool;   // El robot se mueve hacia el buffer
      Mov2 : Bool;   // El robot se mueve hacia la máquina
      Mov3 : Bool;   // El robot vuelve a la posición de reposo
      Act1 : Bool;   // El robot coje una pieza
      Act2 : Bool;   // El robot deja la pieza en maquina
      Wait : Bool;   // El robot espera a que la maquina esté libre
      Aviso_Emergencia : Bool;   // Aviso que indica que se ha activado el estado de emergencia
      STDBY : Bool;   // Standby
   END_VAR
   VAR_IN_OUT
      Aviso_Maquina_Libre : Bool;   // Aviso que le indica al robot que la máquina esta libre
      Aviso_Error_Sincrono : Bool;   // Aviso que indica que ha ocurrido un error relacionado con el tiempo limite
      Aviso_Error_Asincrono : Bool;   // Aviso que indica que ha ocurrido un error NO relacionado con el tiempo(ej: Pinza abierta cuando no deberia)
   END_VAR
   VAR
      BDT : Bool;   // Bit de trabajo
      X_Error_Sincrono : Bool;   // Etapa de error sincrono
      X_Error_Asincrono : Bool;   // Etapa de error asincrono
      X_EMER : Bool;   // Estado de emergencia
      X_REPOSO : Bool;   // Estado de reposo
      X_1_1 : Bool;   // Maniobra 1
      X_1_2 : Bool;   // Maniobra 2
      Aviso_Fin_Maniobra : Bool;   // Aviso que da el robot para indicar que ha terminado la maniobra
      Aviso_Tiempo_Lim : Bool;   // Aviso tiempo limite
      Aviso_Pinza_Abierta : Bool;   // Aviso pinza abierta
      Aviso_No_Pieza : Bool;   // Aviso no pieza
      MOV_Carga : "MOV_BRAZO_1";
      MOV_Descarga : "MOV_BRAZO_2";
   END_VAR
BEGIN

REGION Network 1: EMERGENCIA
   // MAXIMA PRIORIDAD
         A     #EMER;
         S     #X_EMER;

   //ESTADOS
         R     #X_1_1;
         R     #X_1_2;
         R     #X_REPOSO;
         R     #X_Error_Sincrono;
         R     #X_Error_Asincrono;


   //RESET TEMP

         R     #Timer_LIM;
         FR    #Timer_LIM;

         JCN   _EMER;

         CALL  #MOV_Carga
         ( Sensor_Pieza               := ,
           Sensor_Pinza_Llena         := ,
           Sensor_Llegada_a_Buffer    := ,
           Sensor_Llegada_a_Maquina   := ,
           "Sensor_Llegada_a _Reposo" := ,
           EMER                       := TRUE,
           Tiempo_lim                 := #Tiempo_lim,
           Timer_LIM                  := #Timer_LIM,
           MOV1                       := #Mov1,
           MOV2                       := #Mov2,
           MOV3                       := #Mov3,
           ACT1                       := #Act1,
           ACT2                       := #Act2,
           WAIT1                      := #Wait,
           Aviso_Error_Tiempo_Limite  := #Aviso_Tiempo_Lim,
           Aviso_Fin_Maniobra         := #Aviso_Fin_Maniobra,
           Aviso_Error_No_Pieza       := #Aviso_No_Pieza,
           Aviso_Error_Pinza_Abierta  := #Aviso_Pinza_Abierta,
           Aviso_Maquina_Libre        := #Aviso_Maquina_Libre
         );

         CALL  #MOV_Descarga
         ( Sensor_Pieza               := ,
           Sensor_Pinza_Llena         := ,
           Sensor_Llegada_a_Maquina   := ,
           Sensor_Llegada_a_Buffer    := ,
           "Sensor_Llegada_a _Reposo" := ,
           EMER                       := TRUE,
           Tiempo_lim                 := #Tiempo_lim,
           Timer_LIM                  := #Timer_LIM,
           MOV1                       := #Mov1,
           MOV2                       := #Mov2,
           MOV3                       := #Mov3,
           ACT1                       := #Act1,
           ACT2                       := #Act2,
           Aviso_Error_Tiempo_Limite  := #Aviso_Tiempo_Lim,
           Aviso_Fin_Maniobra         := #Aviso_Fin_Maniobra,
           Aviso_Error_No_Pieza       := #Aviso_No_Pieza,
           Aviso_Error_Pinza_Abierta  := #Aviso_Pinza_Abierta
         );



   _EMER:NOP   0;
END_REGION

REGION Network 2: SALIDA DE X_EMER A X_REPOSO
         A     #X_EMER;
         =     #Aviso_Emergencia;

         A     #X_EMER;
         AN    #EMER;
         A     #REARME;
         S     #X_REPOSO;
         R     #X_EMER;


         A     #X_EMER;
         BEC;
END_REGION

REGION Network 3: START===FALSE
         AN    #START;

   //ESTADOS

         R     #BDT;
         R     #X_1_1;
         R     #X_1_2;
         R     #X_REPOSO;
         R     #X_Error_Sincrono;
         R     #X_Error_Asincrono;
         R     #STDBY;

   //RESET TEMP

         R     #Timer_LIM;
         FR    #Timer_LIM;

         JCN   _START_FALSE;

         CALL  #MOV_Carga
         ( Sensor_Pieza               := ,
           Sensor_Pinza_Llena         := ,
           Sensor_Llegada_a_Buffer    := ,
           Sensor_Llegada_a_Maquina   := ,
           "Sensor_Llegada_a _Reposo" := ,
           EMER                       := TRUE,
           Tiempo_lim                 := #Tiempo_lim,
           Timer_LIM                  := #Timer_LIM,
           MOV1                       := #Mov1,
           MOV2                       := #Mov2,
           MOV3                       := #Mov3,
           ACT1                       := #Act1,
           ACT2                       := #Act2,
           WAIT1                      := #Wait,
           Aviso_Error_Tiempo_Limite  := #Aviso_Tiempo_Lim,
           Aviso_Fin_Maniobra         := #Aviso_Fin_Maniobra,
           Aviso_Error_No_Pieza       := #Aviso_No_Pieza,
           Aviso_Error_Pinza_Abierta  := #Aviso_Pinza_Abierta,
           Aviso_Maquina_Libre        := #Aviso_Maquina_Libre
         );

         CALL  #MOV_Descarga
         ( Sensor_Pieza               := ,
           Sensor_Pinza_Llena         := ,
           Sensor_Llegada_a_Maquina   := ,
           Sensor_Llegada_a_Buffer    := ,
           "Sensor_Llegada_a _Reposo" := ,
           EMER                       := TRUE,
           Tiempo_lim                 := #Tiempo_lim,
           Timer_LIM                  := #Timer_LIM,
           MOV1                       := #Mov1,
           MOV2                       := #Mov2,
           MOV3                       := #Mov3,
           ACT1                       := #Act1,
           ACT2                       := #Act2,
           Aviso_Error_Tiempo_Limite  := #Aviso_Tiempo_Lim,
           Aviso_Fin_Maniobra         := #Aviso_Fin_Maniobra,
           Aviso_Error_No_Pieza       := #Aviso_No_Pieza,
           Aviso_Error_Pinza_Abierta  := #Aviso_Pinza_Abierta
         );



   _START_FALSE:NOP   0;

         AN    #START;
         BEC;
END_REGION

REGION Network 4: ERROR_SINCRONO===TRUE
         A     #Aviso_Tiempo_Lim;
         S     #X_Error_Sincrono;
         S     #Aviso_Error_Sincrono;
   //RESETEO UNICAS ETAPAS QUE TIENEN MOVIMIENTOS Y TRATAN CON TIEMPOS
         R     #X_1_1;
         R     #X_1_2;

         JCN   _ERROR_SINCRONO;
         CALL  #MOV_Carga
         ( Sensor_Pieza               := ,
           Sensor_Pinza_Llena         := ,
           Sensor_Llegada_a_Buffer    := ,
           Sensor_Llegada_a_Maquina   := ,
           "Sensor_Llegada_a _Reposo" := ,
           EMER                       := TRUE,
           Tiempo_lim                 := #Tiempo_lim,
           Timer_LIM                  := #Timer_LIM,
           MOV1                       := #Mov1,
           MOV2                       := #Mov2,
           MOV3                       := #Mov3,
           ACT1                       := #Act1,
           ACT2                       := #Act2,
           WAIT1                      := #Wait,
           Aviso_Error_Tiempo_Limite  := #Aviso_Tiempo_Lim,
           Aviso_Fin_Maniobra         := #Aviso_Fin_Maniobra,
           Aviso_Error_No_Pieza       := #Aviso_No_Pieza,
           Aviso_Error_Pinza_Abierta  := #Aviso_Pinza_Abierta,
           Aviso_Maquina_Libre        := #Aviso_Maquina_Libre
         );

         CALL  #MOV_Descarga
         ( Sensor_Pieza               := ,
           Sensor_Pinza_Llena         := ,
           Sensor_Llegada_a_Maquina   := ,
           Sensor_Llegada_a_Buffer    := ,
           "Sensor_Llegada_a _Reposo" := ,
           EMER                       := TRUE,
           Tiempo_lim                 := #Tiempo_lim,
           Timer_LIM                  := #Timer_LIM,
           MOV1                       := #Mov1,
           MOV2                       := #Mov2,
           MOV3                       := #Mov3,
           ACT1                       := #Act1,
           ACT2                       := #Act2,
           Aviso_Error_Tiempo_Limite  := #Aviso_Tiempo_Lim,
           Aviso_Fin_Maniobra         := #Aviso_Fin_Maniobra,
           Aviso_Error_No_Pieza       := #Aviso_No_Pieza,
           Aviso_Error_Pinza_Abierta  := #Aviso_Pinza_Abierta
         );



   _ERROR_SINCRONO:NOP   0;
END_REGION

REGION Network 5: ERROR_ASINCRONO===TRUE
         A     #Aviso_Pinza_Abierta;
         O     #Aviso_No_Pieza;
         S     #X_Error_Asincrono;
         S     #Aviso_Error_Asincrono;

   //RESETEO ETAPAS QUE TIENEN MOVIMIENTOS Y TRATAN CON TIEMPOS
         R     #X_1_1;
         R     #X_1_2;

         JCN   _ERROR_ASINCRONO;

         CALL  #MOV_Carga
         ( Sensor_Pieza               := ,
           Sensor_Pinza_Llena         := ,
           Sensor_Llegada_a_Buffer    := ,
           Sensor_Llegada_a_Maquina   := ,
           "Sensor_Llegada_a _Reposo" := ,
           EMER                       := TRUE,
           Tiempo_lim                 := #Tiempo_lim,
           Timer_LIM                  := #Timer_LIM,
           MOV1                       := #Mov1,
           MOV2                       := #Mov2,
           MOV3                       := #Mov3,
           ACT1                       := #Act1,
           ACT2                       := #Act2,
           WAIT1                      := #Wait,
           Aviso_Error_Tiempo_Limite  := #Aviso_Tiempo_Lim,
           Aviso_Fin_Maniobra         := #Aviso_Fin_Maniobra,
           Aviso_Error_No_Pieza       := #Aviso_No_Pieza,
           Aviso_Error_Pinza_Abierta  := #Aviso_Pinza_Abierta,
           Aviso_Maquina_Libre        := #Aviso_Maquina_Libre
         );

